LIN {X 0.007,Y -350.625,Z 530.640,A 0.000,B 0.000,C 90.000,E1 115.155} C_DIS
LIN {X -0.166,Y -363.454,Z 530.626,A 0.000,B 0.000,C 90.000,E1 112.770} C_DIS
LIN {X 0.046,Y -377.608,Z 530.613,A 0.000,B 0.000,C 90.000,E1 110.375} C_DIS
LIN {X 0.134,Y -393.193,Z 530.600,A 0.000,B 0.000,C 90.000,E1 108.055} C_DIS
LIN {X -0.144,Y -410.320,Z 530.588,A 0.000,B 0.000,C 90.000,E1 105.843} C_DIS
LIN {X -0.125,Y -429.118,Z 530.576,A 0.000,B 0.000,C 90.000,E1 103.647} C_DIS
LIN {X 0.160,Y -449.156,Z 530.564,A 0.000,B 0.000,C 90.000,E1 101.535} C_DIS
LIN {X -0.139,Y -469.752,Z 530.554,A 0.000,B 0.000,C 90.000,E1 99.670} C_DIS
LIN {X 0.073,Y -477.496,Z 530.550,A 0.000,B 0.000,C 90.000,E1 98.973} C_DIS
LIN {X 0.123,Y -479.452,Z 530.549,A 0.000,B 0.000,C 90.000,E1 98.746} C_DIS
LIN {X -0.005,Y -481.138,Z 530.547,A 0.000,B 0.000,C 90.000,E1 98.511} C_DIS
LIN {X -0.136,Y -482.404,Z 530.546,A 0.000,B 0.000,C 90.000,E1 98.276} C_DIS
LIN {X 0.031,Y -483.966,Z 530.543,A 0.000,B 0.000,C 90.000,E1 97.757} C_DIS
LIN {X 0.207,Y -484.472,Z 530.540,A 0.000,B 0.000,C 90.000,E1 97.239} C_DIS
LIN {X -0.087,Y -484.003,Z 530.538,A 0.000,B 0.000,C 90.000,E1 96.777} C_DIS
LIN {X 0.102,Y -482.486,Z 530.535,A 0.000,B 0.000,C 90.000,E1 96.258} C_DIS
LIN {X -0.070,Y -481.251,Z 530.533,A 0.000,B 0.000,C 90.000,E1 96.030} C_DIS
LIN {X -0.191,Y -479.606,Z 530.532,A 0.000,B 0.000,C 90.000,E1 95.796} C_DIS
LIN {X 0.087,Y -461.916,Z 530.519,A 0.000,B 0.000,C 90.000,E1 93.498} C_DIS
LIN {X 0.151,Y -451.298,Z 530.511,A 0.000,B 0.000,C 90.000,E1 91.949} C_DIS
LIN {X -0.041,Y -438.774,Z 530.499,A 0.000,B 0.000,C 90.000,E1 89.885} C_DIS
LIN {X 0.054,Y -429.143,Z 530.490,A 0.000,B 0.000,C 90.000,E1 88.282} C_DIS
LIN {X -0.197,Y -416.360,Z 530.479,A 0.000,B 0.000,C 90.000,E1 86.159} C_DIS
LIN {X 0.150,Y -403.728,Z 530.466,A 0.000,B 0.000,C 90.000,E1 83.913} C_DIS
LIN {X 0.177,Y -392.888,Z 530.455,A 0.000,B 0.000,C 90.000,E1 81.951} C_DIS
LIN {X 0.024,Y -381.992,Z 530.444,A 0.000,B 0.000,C 90.000,E1 79.982} C_DIS
LIN {X 0.133,Y -366.500,Z 530.428,A 0.000,B 0.000,C 90.000,E1 77.061} C_DIS
LIN {X 0.143,Y -357.922,Z 530.418,A 0.000,B 0.000,C 90.000,E1 75.283} C_DIS
LIN {X -0.016,Y -346.420,Z 530.403,A 0.000,B 0.000,C 90.000,E1 72.598} C_DIS
LIN {X 0.049,Y -335.338,Z 530.386,A 0.000,B 0.000,C 90.000,E1 69.518} C_DIS
LIN {X -0.030,Y -325.168,Z 530.369,A 0.000,B 0.000,C 90.000,E1 66.410} C_DIS
LIN {X -0.152,Y -317.591,Z 530.355,A 0.000,B 0.000,C 90.000,E1 63.896} C_DIS
LIN {X -0.045,Y -309.997,Z 530.341,A 0.000,B 0.000,C 90.000,E1 61.307} C_DIS
LIN {X 0.168,Y -302.402,Z 530.326,A 0.000,B 0.000,C 90.000,E1 58.663} C_DIS
LIN {X 0.004,Y -293.272,Z 530.308,A 0.000,B 0.000,C 90.000,E1 55.388} C_DIS
LIN {X -0.063,Y -286.330,Z 530.293,A 0.000,B 0.000,C 90.000,E1 52.718} C_DIS
LIN {X -0.042,Y -281.026,Z 530.281,A 0.000,B 0.000,C 90.000,E1 50.678} C_DIS
LIN {X 0.012,Y -277.267,Z 530.274,A 0.000,B 0.000,C 90.000,E1 49.299} C_DIS
LIN {X 0.024,Y -273.186,Z 530.266,A 0.000,B 0.000,C 90.000,E1 47.919} C_DIS
LIN {X 0.128,Y -266.584,Z 530.255,A 0.000,B 0.000,C 90.000,E1 45.810} C_DIS
LIN {X 0.076,Y -259.610,Z 530.243,A 0.000,B 0.000,C 90.000,E1 43.704} C_DIS
LIN {X 0.135,Y -249.136,Z 530.225,A 0.000,B 0.000,C 90.000,E1 40.458} C_DIS
LIN {X -0.025,Y -239.322,Z 530.207,A 0.000,B 0.000,C 90.000,E1 37.202} C_DIS
LIN {X 0.076,Y -231.432,Z 530.190,A 0.000,B 0.000,C 90.000,E1 34.199} C_DIS
LIN {X -0.073,Y -224.272,Z 530.173,A 0.000,B 0.000,C 90.000,E1 31.209} C_DIS
LIN {X 0.064,Y -217.981,Z 530.156,A 0.000,B 0.000,C 90.000,E1 28.103} C_DIS
LIN {X -0.070,Y -212.533,Z 530.139,A 0.000,B 0.000,C 90.000,E1 25.027} C_DIS
LIN {X 0.062,Y -207.862,Z 530.121,A 0.000,B 0.000,C 90.000,E1 21.844} C_DIS
LIN {X 0.037,Y -203.164,Z 530.099,A 0.000,B 0.000,C 90.000,E1 17.873} C_DIS
LIN {X -0.011,Y -198.859,Z 530.073,A 0.000,B 0.000,C 90.000,E1 13.063} C_DIS
LIN {X 0.096,Y -195.722,Z 530.041,A 0.000,B 0.000,C 90.000,E1 7.352} C_DIS
LIN {X 0.022,Y -196.744,Z 529.961,A 0.000,B 0.000,C 90.000,E1 352.996} C_DIS
LIN {X 0.044,Y -199.908,Z 529.934,A 0.000,B 0.000,C 90.000,E1 348.117} C_DIS
LIN {X -0.099,Y -204.347,Z 529.907,A 0.000,B 0.000,C 90.000,E1 343.323} C_DIS
LIN {X -0.047,Y -208.988,Z 529.885,A 0.000,B 0.000,C 90.000,E1 339.316} C_DIS
LIN {X -0.013,Y -214.345,Z 529.863,A 0.000,B 0.000,C 90.000,E1 335.357} C_DIS
LIN {X 0.053,Y -220.253,Z 529.841,A 0.000,B 0.000,C 90.000,E1 331.435} C_DIS
LIN {X 0.050,Y -226.713,Z 529.820,A 0.000,B 0.000,C 90.000,E1 327.582} C_DIS
LIN {X 0.037,Y -233.852,Z 529.799,A 0.000,B 0.000,C 90.000,E1 323.783} C_DIS
LIN {X -0.099,Y -241.522,Z 529.778,A 0.000,B 0.000,C 90.000,E1 320.070} C_DIS
LIN {X -0.078,Y -250.132,Z 529.758,A 0.000,B 0.000,C 90.000,E1 316.377} C_DIS
LIN {X -0.146,Y -259.993,Z 529.737,A 0.000,B 0.000,C 90.000,E1 312.771} C_DIS
LIN {X -0.008,Y -271.110,Z 529.718,A 0.000,B 0.000,C 90.000,E1 309.197} C_DIS
LIN {X 0.019,Y -283.470,Z 529.698,A 0.000,B 0.000,C 90.000,E1 305.724} C_DIS
LIN {X 0.018,Y -297.205,Z 529.680,A 0.000,B 0.000,C 90.000,E1 302.339} C_DIS
LIN {X 0.091,Y -312.087,Z 529.661,A 0.000,B 0.000,C 90.000,E1 299.027} C_DIS
LIN {X -0.031,Y -326.602,Z 529.645,A 0.000,B 0.000,C 90.000,E1 296.155} C_DIS
LIN {X -0.104,Y -335.578,Z 529.637,A 0.000,B 0.000,C 90.000,E1 294.591} C_DIS
LIN {X -0.001,Y -349.328,Z 529.625,A 0.000,B 0.000,C 90.000,E1 292.408} C_DIS
LIN {X -0.061,Y -364.291,Z 529.613,A 0.000,B 0.000,C 90.000,E1 290.301} C_DIS
LIN {X 0.072,Y -385.334,Z 529.598,A 0.000,B 0.000,C 90.000,E1 287.638} C_DIS
LIN {X -0.069,Y -402.321,Z 529.587,A 0.000,B 0.000,C 90.000,E1 285.662} C_DIS
LIN {X -0.186,Y -417.218,Z 529.578,A 0.000,B 0.000,C 90.000,E1 284.008} C_DIS
LIN {X -0.176,Y -429.390,Z 529.570,A 0.000,B 0.000,C 90.000,E1 282.647} C_DIS
LIN {X -0.114,Y -441.000,Z 529.563,A 0.000,B 0.000,C 90.000,E1 281.299} C_DIS
LIN {X 0.019,Y -447.666,Z 529.558,A 0.000,B 0.000,C 90.000,E1 280.489} C_DIS
LIN {X 0.026,Y -455.859,Z 529.552,A 0.000,B 0.000,C 90.000,E1 279.443} C_DIS
LIN {X 0.132,Y -463.364,Z 529.547,A 0.000,B 0.000,C 90.000,E1 278.398} C_DIS
LIN {X 0.017,Y -468.372,Z 529.542,A 0.000,B 0.000,C 90.000,E1 277.644} C_DIS
LIN {X -0.052,Y -472.900,Z 529.538,A 0.000,B 0.000,C 90.000,E1 276.891} C_DIS
LIN {X -0.144,Y -476.941,Z 529.534,A 0.000,B 0.000,C 90.000,E1 276.144} C_DIS
LIN {X -0.146,Y -480.361,Z 529.530,A 0.000,B 0.000,C 90.000,E1 275.391} C_DIS
LIN {X -0.171,Y -483.141,Z 529.526,A 0.000,B 0.000,C 90.000,E1 274.645} C_DIS
LIN {X -0.039,Y -484.544,Z 529.523,A 0.000,B 0.000,C 90.000,E1 274.131} C_DIS
LIN {X 0.140,Y -485.652,Z 529.520,A 0.000,B 0.000,C 90.000,E1 273.612} C_DIS
LIN {X -0.161,Y -486.454,Z 529.517,A 0.000,B 0.000,C 90.000,E1 273.151} C_DIS
LIN {X 0.002,Y -486.937,Z 529.515,A 0.000,B 0.000,C 90.000,E1 272.636} C_DIS
LIN {X 0.173,Y -487.084,Z 529.512,A 0.000,B 0.000,C 90.000,E1 272.121} C_DIS
LIN {X -0.122,Y -486.839,Z 529.509,A 0.000,B 0.000,C 90.000,E1 271.661} C_DIS
LIN {X 0.053,Y -486.202,Z 529.506,A 0.000,B 0.000,C 90.000,E1 271.146} C_DIS
LIN {X 0.229,Y -485.150,Z 529.504,A 0.000,B 0.000,C 90.000,E1 270.630} C_DIS
LIN {X -0.084,Y -483.586,Z 529.501,A 0.000,B 0.000,C 90.000,E1 270.172} C_DIS
LIN {X 0.082,Y -481.379,Z 529.498,A 0.000,B 0.000,C 90.000,E1 269.656} C_DIS
LIN {X 0.231,Y -478.423,Z 529.495,A 0.000,B 0.000,C 90.000,E1 269.141} C_DIS
LIN {X -0.113,Y -474.579,Z 529.493,A 0.000,B 0.000,C 90.000,E1 268.682} C_DIS
LIN {X 0.015,Y -469.635,Z 529.490,A 0.000,B 0.000,C 90.000,E1 268.165} C_DIS
LIN {X -0.092,Y -466.805,Z 529.488,A 0.000,B 0.000,C 90.000,E1 267.936} C_DIS
LIN {X -0.197,Y -463.629,Z 529.487,A 0.000,B 0.000,C 90.000,E1 267.707} C_DIS
LIN {X -0.022,Y -460.564,Z 529.486,A 0.000,B 0.000,C 90.000,E1 267.478} C_DIS
LIN {X 0.152,Y -453.814,Z 529.484,A 0.000,B 0.000,C 90.000,E1 267.078} C_DIS
LIN {X -0.011,Y -446.799,Z 529.482,A 0.000,B 0.000,C 90.000,E1 266.788} C_DIS
LIN {X -0.202,Y -439.772,Z 529.481,A 0.000,B 0.000,C 90.000,E1 266.560} C_DIS
LIN {X -0.051,Y -432.358,Z 529.480,A 0.000,B 0.000,C 90.000,E1 266.331} C_DIS
LIN {X 0.005,Y -424.212,Z 529.479,A 0.000,B 0.000,C 90.000,E1 266.159} C_DIS
LIN {X -0.004,Y -414.402,Z 529.478,A 0.000,B 0.000,C 90.000,E1 266.045} C_DIS
LIN {X 0.134,Y -407.149,Z 529.478,A 0.000,B 0.000,C 90.000,E1 265.988} C_DIS
LIN {X 0.040,Y -180.920,Z 529.478,A 0.000,B 0.000,C 90.000,E1 265.988} C_DIS
LIN {X -0.084,Y -180.857,Z 529.472,A 0.000,B 0.000,C 90.000,E1 265.008} C_DIS
LIN {X -0.005,Y -178.910,Z 529.443,A 0.000,B 0.000,C 90.000,E1 259.746} C_DIS
LIN {X 0.076,Y -175.954,Z 529.415,A 0.000,B 0.000,C 90.000,E1 254.629} C_DIS
LIN {X 0.022,Y -175.423,Z 529.410,A 0.000,B 0.000,C 90.000,E1 253.795} C_DIS
LIN {X 0.025,Y -172.184,Z 529.386,A 0.000,B 0.000,C 90.000,E1 249.518} C_DIS
LIN {X 0.063,Y -171.656,Z 529.381,A 0.000,B 0.000,C 90.000,E1 248.646} C_DIS
LIN {X 0.057,Y -167.880,Z 529.357,A 0.000,B 0.000,C 90.000,E1 244.332} C_DIS
LIN {X 0.001,Y -166.615,Z 529.348,A 0.000,B 0.000,C 90.000,E1 242.615} C_DIS
LIN {X -0.006,Y -162.602,Z 529.324,A 0.000,B 0.000,C 90.000,E1 238.250} C_DIS
LIN {X -0.032,Y -161.288,Z 529.314,A 0.000,B 0.000,C 90.000,E1 236.501} C_DIS
LIN {X 0.003,Y -157.287,Z 529.289,A 0.000,B 0.000,C 90.000,E1 232.065} C_DIS
LIN {X 0.026,Y -156.004,Z 529.279,A 0.000,B 0.000,C 90.000,E1 230.275} C_DIS
LIN {X -0.014,Y -152.262,Z 529.254,A 0.000,B 0.000,C 90.000,E1 225.810} C_DIS
LIN {X 0.008,Y -150.500,Z 529.239,A 0.000,B 0.000,C 90.000,E1 223.095} C_DIS
LIN {X 0.038,Y -147.224,Z 529.214,A 0.000,B 0.000,C 90.000,E1 218.543} C_DIS
LIN {X 0.008,Y -145.247,Z 529.194,A 0.000,B 0.000,C 90.000,E1 214.898} C_DIS
LIN {X -0.076,Y -142.364,Z 529.163,A 0.000,B 0.000,C 90.000,E1 209.411} C_DIS
LIN {X 0.045,Y -141.750,Z 529.153,A 0.000,B 0.000,C 90.000,E1 207.513} C_DIS
LIN {X -0.029,Y -139.494,Z 529.117,A 0.000,B 0.000,C 90.000,E1 201.046} C_DIS
LIN {X 0.007,Y -138.997,Z 529.101,A 0.000,B 0.000,C 90.000,E1 198.236} C_DIS
LIN {X -0.036,Y -138.338,Z 529.055,A 0.000,B 0.000,C 90.000,E1 189.849} C_DIS
LIN {X -0.014,Y -139.412,Z 529.008,A 0.000,B 0.000,C 90.000,E1 181.432} C_DIS
LIN {X 0.040,Y -141.325,Z 528.972,A 0.000,B 0.000,C 90.000,E1 174.894} C_DIS
LIN {X -0.003,Y -142.683,Z 528.956,A 0.000,B 0.000,C 90.000,E1 172.129} C_DIS
LIN {X -0.024,Y -145.042,Z 528.931,A 0.000,B 0.000,C 90.000,E1 167.521} C_DIS
LIN {X -0.026,Y -147.667,Z 528.910,A 0.000,B 0.000,C 90.000,E1 163.850} C_DIS
LIN {X 0.009,Y -150.309,Z 528.890,A 0.000,B 0.000,C 90.000,E1 160.188} C_DIS
LIN {X 0.020,Y -153.720,Z 528.870,A 0.000,B 0.000,C 90.000,E1 156.561} C_DIS
LIN {X -0.067,Y -157.134,Z 528.850,A 0.000,B 0.000,C 90.000,E1 152.999} C_DIS
LIN {X 0.009,Y -161.281,Z 528.830,A 0.000,B 0.000,C 90.000,E1 149.410} C_DIS
LIN {X 0.026,Y -164.397,Z 528.815,A 0.000,B 0.000,C 90.000,E1 146.755} C_DIS
LIN {X 0.023,Y -169.076,Z 528.796,A 0.000,B 0.000,C 90.000,E1 143.256} C_DIS
LIN {X -0.026,Y -171.634,Z 528.786,A 0.000,B 0.000,C 90.000,E1 141.537} C_DIS
LIN {X 0.021,Y -176.595,Z 528.767,A 0.000,B 0.000,C 90.000,E1 138.081} C_DIS
LIN {X -0.107,Y -180.893,Z 528.753,A 0.000,B 0.000,C 90.000,E1 135.567} C_DIS
LIN {X 0.015,Y -186.308,Z 528.734,A 0.000,B 0.000,C 90.000,E1 132.162} C_DIS
LIN {X 0.076,Y -191.412,Z 528.719,A 0.000,B 0.000,C 90.000,E1 129.358} C_DIS
LIN {X -0.043,Y -192.207,Z 528.716,A 0.000,B 0.000,C 90.000,E1 128.910} C_DIS
LIN {X -0.099,Y -289.108,Z 528.716,A 0.000,B 0.000,C 90.000,E1 128.910} C_DIS
LIN {X 0.061,Y -291.712,Z 528.716,A 0.000,B 0.000,C 90.000,E1 128.830} C_DIS
LIN {X 0.026,Y -294.579,Z 528.715,A 0.000,B 0.000,C 90.000,E1 128.705} C_DIS
LIN {X 0.024,Y -298.101,Z 528.713,A 0.000,B 0.000,C 90.000,E1 128.418} C_DIS
LIN {X 0.036,Y -301.731,Z 528.711,A 0.000,B 0.000,C 90.000,E1 127.935} C_DIS
LIN {X 0.036,Y -303.492,Z 528.709,A 0.000,B 0.000,C 90.000,E1 127.604} C_DIS
LIN {X -0.022,Y -304.870,Z 528.707,A 0.000,B 0.000,C 90.000,E1 127.282} C_DIS
LIN {X -0.001,Y -310.679,Z 528.696,A 0.000,B 0.000,C 90.000,E1 125.311} C_DIS
LIN {X -0.024,Y -321.264,Z 528.678,A 0.000,B 0.000,C 90.000,E1 122.084} C_DIS
LIN {X 0.130,Y -332.150,Z 528.662,A 0.000,B 0.000,C 90.000,E1 119.205} C_DIS
LIN {X -0.051,Y -344.433,Z 528.647,A 0.000,B 0.000,C 90.000,E1 116.437} C_DIS
LIN {X -0.082,Y -356.610,Z 528.633,A 0.000,B 0.000,C 90.000,E1 114.003} C_DIS
LIN {X 0.082,Y -370.065,Z 528.620,A 0.000,B 0.000,C 90.000,E1 111.589} C_DIS
LIN {X -0.022,Y -384.893,Z 528.607,A 0.000,B 0.000,C 90.000,E1 109.268} C_DIS
LIN {X -0.005,Y -401.205,Z 528.594,A 0.000,B 0.000,C 90.000,E1 106.985} C_DIS
LIN {X -0.087,Y -419.119,Z 528.582,A 0.000,B 0.000,C 90.000,E1 104.773} C_DIS
LIN {X 0.140,Y -438.656,Z 528.570,A 0.000,B 0.000,C 90.000,E1 102.591} C_DIS
LIN {X 0.136,Y -458.972,Z 528.559,A 0.000,B 0.000,C 90.000,E1 100.602} C_DIS
LIN {X -0.122,Y -477.137,Z 528.550,A 0.000,B 0.000,C 90.000,E1 99.029} C_DIS
LIN {X -0.077,Y -479.223,Z 528.549,A 0.000,B 0.000,C 90.000,E1 98.803} C_DIS
LIN {X -0.207,Y -481.005,Z 528.547,A 0.000,B 0.000,C 90.000,E1 98.568} C_DIS
LIN {X 0.138,Y -482.344,Z 528.546,A 0.000,B 0.000,C 90.000,E1 98.276} C_DIS
LIN {X -0.175,Y -484.021,Z 528.543,A 0.000,B 0.000,C 90.000,E1 97.814} C_DIS
LIN {X 0.001,Y -484.625,Z 528.541,A 0.000,B 0.000,C 90.000,E1 97.296} C_DIS
LIN {X 0.187,Y -484.254,Z 528.538,A 0.000,B 0.000,C 90.000,E1 96.777} C_DIS
LIN {X -0.104,Y -482.849,Z 528.535,A 0.000,B 0.000,C 90.000,E1 96.315} C_DIS
LIN {X 0.203,Y -481.685,Z 528.534,A 0.000,B 0.000,C 90.000,E1 96.030} C_DIS
LIN {X 0.083,Y -480.128,Z 528.532,A 0.000,B 0.000,C 90.000,E1 95.796} C_DIS
LIN {X 0.157,Y -460.553,Z 528.518,A 0.000,B 0.000,C 90.000,E1 93.269} C_DIS
LIN {X 0.212,Y -450.047,Z 528.510,A 0.000,B 0.000,C 90.000,E1 91.718} C_DIS
LIN {X -0.201,Y -439.126,Z 528.500,A 0.000,B 0.000,C 90.000,E1 89.943} C_DIS
LIN {X 0.063,Y -427.874,Z 528.489,A 0.000,B 0.000,C 90.000,E1 88.051} C_DIS
LIN {X 0.210,Y -415.100,Z 528.477,A 0.000,B 0.000,C 90.000,E1 85.869} C_DIS
LIN {X 0.079,Y -402.485,Z 528.465,A 0.000,B 0.000,C 90.000,E1 83.685} C_DIS
LIN {X 0.071,Y -391.630,Z 528.454,A 0.000,B 0.000,C 90.000,E1 81.724} C_DIS
LIN {X -0.040,Y -380.732,Z 528.443,A 0.000,B 0.000,C 90.000,E1 79.746} C_DIS
LIN {X 0.078,Y -362.338,Z 528.424,A 0.000,B 0.000,C 90.000,E1 76.228} C_DIS
LIN {X -0.096,Y -351.588,Z 528.410,A 0.000,B 0.000,C 90.000,E1 73.866} C_DIS
LIN {X 0.089,Y -343.134,Z 528.398,A 0.000,B 0.000,C 90.000,E1 71.710} C_DIS
LIN {X -0.041,Y -331.364,Z 528.380,A 0.000,B 0.000,C 90.000,E1 68.337} C_DIS
LIN {X 0.060,Y -321.469,Z 528.362,A 0.000,B 0.000,C 90.000,E1 65.177} C_DIS
LIN {X 0.116,Y -315.842,Z 528.352,A 0.000,B 0.000,C 90.000,E1 63.256} C_DIS
LIN {X -0.099,Y -308.215,Z 528.337,A 0.000,B 0.000,C 90.000,E1 60.717} C_DIS
LIN {X 0.065,Y -300.615,Z 528.323,A 0.000,B 0.000,C 90.000,E1 58.074} C_DIS
LIN {X 0.007,Y -291.582,Z 528.304,A 0.000,B 0.000,C 90.000,E1 54.769} C_DIS
LIN {X 0.066,Y -284.646,Z 528.289,A 0.000,B 0.000,C 90.000,E1 52.065} C_DIS
LIN {X 0.015,Y -279.246,Z 528.278,A 0.000,B 0.000,C 90.000,E1 50.033} C_DIS
LIN {X -0.127,Y -275.337,Z 528.270,A 0.000,B 0.000,C 90.000,E1 48.690} C_DIS
LIN {X -0.137,Y -271.113,Z 528.263,A 0.000,B 0.000,C 90.000,E1 47.310} C_DIS
LIN {X -0.143,Y -265.514,Z 528.253,A 0.000,B 0.000,C 90.000,E1 45.567} C_DIS
LIN {X -0.021,Y -258.491,Z 528.241,A 0.000,B 0.000,C 90.000,E1 43.419} C_DIS
LIN {X 0.022,Y -248.070,Z 528.223,A 0.000,B 0.000,C 90.000,E1 40.172} C_DIS
LIN {X 0.036,Y -239.368,Z 528.207,A 0.000,B 0.000,C 90.000,E1 37.237} C_DIS
LIN {X -0.045,Y -231.492,Z 528.190,A 0.000,B 0.000,C 90.000,E1 34.278} C_DIS
LIN {X -0.069,Y -224.332,Z 528.174,A 0.000,B 0.000,C 90.000,E1 31.258} C_DIS
LIN {X 0.064,Y -218.015,Z 528.156,A 0.000,B 0.000,C 90.000,E1 28.153} C_DIS
LIN {X -0.076,Y -212.566,Z 528.139,A 0.000,B 0.000,C 90.000,E1 25.079} C_DIS
LIN {X 0.053,Y -207.885,Z 528.122,A 0.000,B 0.000,C 90.000,E1 21.897} C_DIS
LIN {X -0.038,Y -203.189,Z 528.100,A 0.000,B 0.000,C 90.000,E1 17.946} C_DIS
LIN {X -0.027,Y -198.863,Z 528.073,A 0.000,B 0.000,C 90.000,E1 13.119} C_DIS
LIN {X 0.077,Y -195.705,Z 528.041,A 0.000,B 0.000,C 90.000,E1 7.409} C_DIS
LIN {X 0.019,Y -196.653,Z 527.961,A 0.000,B 0.000,C 90.000,E1 352.996} C_DIS
LIN {X 0.037,Y -199.811,Z 527.934,A 0.000,B 0.000,C 90.000,E1 348.117} C_DIS
LIN {X -0.110,Y -204.250,Z 527.907,A 0.000,B 0.000,C 90.000,E1 343.323} C_DIS
LIN {X -0.061,Y -208.893,Z 527.885,A 0.000,B 0.000,C 90.000,E1 339.316} C_DIS
LIN {X -0.031,Y -214.236,Z 527.863,A 0.000,B 0.000,C 90.000,E1 335.357} C_DIS
LIN {X 0.031,Y -220.166,Z 527.841,A 0.000,B 0.000,C 90.000,E1 331.435} C_DIS
LIN {X 0.026,Y -226.620,Z 527.820,A 0.000,B 0.000,C 90.000,E1 327.582} C_DIS
LIN {X 0.010,Y -233.769,Z 527.799,A 0.000,B 0.000,C 90.000,E1 323.783} C_DIS
LIN {X 0.024,Y -241.448,Z 527.778,A 0.000,B 0.000,C 90.000,E1 320.033} C_DIS
LIN {X -0.113,Y -250.080,Z 527.758,A 0.000,B 0.000,C 90.000,E1 316.377} C_DIS
LIN {X -0.023,Y -258.919,Z 527.739,A 0.000,B 0.000,C 90.000,E1 313.095} C_DIS
LIN {X -0.121,Y -269.921,Z 527.720,A 0.000,B 0.000,C 90.000,E1 309.564} C_DIS
LIN {X -0.136,Y -282.164,Z 527.700,A 0.000,B 0.000,C 90.000,E1 306.091} C_DIS
LIN {X -0.019,Y -295.786,Z 527.682,A 0.000,B 0.000,C 90.000,E1 302.673} C_DIS
LIN {X 0.155,Y -310.524,Z 527.663,A 0.000,B 0.000,C 90.000,E1 299.333} C_DIS
LIN {X -0.080,Y -326.591,Z 527.645,A 0.000,B 0.000,C 90.000,E1 296.155} C_DIS
LIN {X -0.154,Y -335.584,Z 527.636,A 0.000,B 0.000,C 90.000,E1 294.591} C_DIS
LIN {X 0.095,Y -351.378,Z 527.623,A 0.000,B 0.000,C 90.000,E1 292.078} C_DIS
LIN {X -0.046,Y -366.538,Z 527.611,A 0.000,B 0.000,C 90.000,E1 289.993} C_DIS
LIN {X 0.026,Y -387.760,Z 527.596,A 0.000,B 0.000,C 90.000,E1 287.347} C_DIS
LIN {X -0.051,Y -404.810,Z 527.585,A 0.000,B 0.000,C 90.000,E1 285.371} C_DIS
LIN {X -0.018,Y -419.735,Z 527.576,A 0.000,B 0.000,C 90.000,E1 283.703} C_DIS
LIN {X 0.043,Y -431.720,Z 527.569,A 0.000,B 0.000,C 90.000,E1 282.355} C_DIS
LIN {X 0.154,Y -443.239,Z 527.561,A 0.000,B 0.000,C 90.000,E1 281.007} C_DIS
LIN {X -0.137,Y -449.792,Z 527.557,A 0.000,B 0.000,C 90.000,E1 280.254} C_DIS
LIN {X -0.108,Y -457.858,Z 527.551,A 0.000,B 0.000,C 90.000,E1 279.208} C_DIS
LIN {X 0.191,Y -463.412,Z 527.547,A 0.000,B 0.000,C 90.000,E1 278.398} C_DIS
LIN {X 0.078,Y -468.442,Z 527.543,A 0.000,B 0.000,C 90.000,E1 277.644} C_DIS
LIN {X -0.203,Y -474.387,Z 527.537,A 0.000,B 0.000,C 90.000,E1 276.663} C_DIS
LIN {X 0.249,Y -478.248,Z 527.533,A 0.000,B 0.000,C 90.000,E1 275.853} C_DIS
LIN {X 0.210,Y -481.467,Z 527.529,A 0.000,B 0.000,C 90.000,E1 275.106} C_DIS
LIN {X -0.107,Y -483.226,Z 527.526,A 0.000,B 0.000,C 90.000,E1 274.645} C_DIS
LIN {X 0.026,Y -484.669,Z 527.523,A 0.000,B 0.000,C 90.000,E1 274.131} C_DIS
LIN {X 0.206,Y -485.766,Z 527.520,A 0.000,B 0.000,C 90.000,E1 273.612} C_DIS
LIN {X -0.122,Y -486.559,Z 527.517,A 0.000,B 0.000,C 90.000,E1 273.154} C_DIS
LIN {X 0.069,Y -487.048,Z 527.515,A 0.000,B 0.000,C 90.000,E1 272.636} C_DIS
LIN {X -0.245,Y -487.209,Z 527.512,A 0.000,B 0.000,C 90.000,E1 272.178} C_DIS
LIN {X -0.054,Y -486.949,Z 527.509,A 0.000,B 0.000,C 90.000,E1 271.661} C_DIS
LIN {X 0.123,Y -486.313,Z 527.506,A 0.000,B 0.000,C 90.000,E1 271.146} C_DIS
LIN {X -0.188,Y -485.245,Z 527.504,A 0.000,B 0.000,C 90.000,E1 270.688} C_DIS
LIN {X -0.014,Y -483.677,Z 527.501,A 0.000,B 0.000,C 90.000,E1 270.172} C_DIS
LIN {X 0.152,Y -481.499,Z 527.498,A 0.000,B 0.000,C 90.000,E1 269.656} C_DIS
LIN {X -0.177,Y -478.524,Z 527.495,A 0.000,B 0.000,C 90.000,E1 269.198} C_DIS
LIN {X 0.129,Y -476.771,Z 527.494,A 0.000,B 0.000,C 90.000,E1 268.912} C_DIS
LIN {X -0.221,Y -472.351,Z 527.491,A 0.000,B 0.000,C 90.000,E1 268.453} C_DIS
LIN {X 0.085,Y -469.779,Z 527.490,A 0.000,B 0.000,C 90.000,E1 268.165} C_DIS
LIN {X -0.032,Y -466.971,Z 527.489,A 0.000,B 0.000,C 90.000,E1 267.936} C_DIS
LIN {X -0.147,Y -463.777,Z 527.487,A 0.000,B 0.000,C 90.000,E1 267.707} C_DIS
LIN {X 0.200,Y -457.215,Z 527.485,A 0.000,B 0.000,C 90.000,E1 267.249} C_DIS
LIN {X 0.153,Y -450.105,Z 527.483,A 0.000,B 0.000,C 90.000,E1 266.906} C_DIS
LIN {X -0.191,Y -443.079,Z 527.481,A 0.000,B 0.000,C 90.000,E1 266.674} C_DIS
LIN {X -0.192,Y -435.942,Z 527.480,A 0.000,B 0.000,C 90.000,E1 266.445} C_DIS
LIN {X 0.123,Y -428.327,Z 527.479,A 0.000,B 0.000,C 90.000,E1 266.216} C_DIS
LIN {X -0.083,Y -419.441,Z 527.478,A 0.000,B 0.000,C 90.000,E1 266.102} C_DIS
LIN {X 0.142,Y -408.334,Z 527.478,A 0.000,B 0.000,C 90.000,E1 265.988} C_DIS
LIN {X 0.095,Y -405.887,Z 527.478,A 0.000,B 0.000,C 90.000,E1 265.988} C_DIS
LIN {X 0.023,Y -180.920,Z 527.478,A 0.000,B 0.000,C 90.000,E1 265.988} C_DIS
LIN {X 0.080,Y -180.856,Z 527.472,A 0.000,B 0.000,C 90.000,E1 264.951} C_DIS
LIN {X -0.021,Y -178.908,Z 527.443,A 0.000,B 0.000,C 90.000,E1 259.746} C_DIS
LIN {X 0.060,Y -175.952,Z 527.415,A 0.000,B 0.000,C 90.000,E1 254.629} C_DIS
LIN {X 0.006,Y -175.418,Z 527.410,A 0.000,B 0.000,C 90.000,E1 253.795} C_DIS
LIN {X 0.008,Y -172.180,Z 527.386,A 0.000,B 0.000,C 90.000,E1 249.518} C_DIS
LIN {X 0.048,Y -171.651,Z 527.381,A 0.000,B 0.000,C 90.000,E1 248.646} C_DIS
LIN {X 0.042,Y -167.876,Z 527.357,A 0.000,B 0.000,C 90.000,E1 244.332} C_DIS
LIN {X -0.015,Y -166.611,Z 527.348,A 0.000,B 0.000,C 90.000,E1 242.615} C_DIS
LIN {X -0.021,Y -162.599,Z 527.324,A 0.000,B 0.000,C 90.000,E1 238.250} C_DIS
LIN {X -0.047,Y -161.283,Z 527.314,A 0.000,B 0.000,C 90.000,E1 236.501} C_DIS
LIN {X -0.012,Y -157.282,Z 527.289,A 0.000,B 0.000,C 90.000,E1 232.065} C_DIS
LIN {X 0.011,Y -156.000,Z 527.279,A 0.000,B 0.000,C 90.000,E1 230.275} C_DIS
LIN {X -0.029,Y -152.258,Z 527.254,A 0.000,B 0.000,C 90.000,E1 225.810} C_DIS
LIN {X -0.006,Y -150.496,Z 527.239,A 0.000,B 0.000,C 90.000,E1 223.095} C_DIS
LIN {X 0.024,Y -147.221,Z 527.214,A 0.000,B 0.000,C 90.000,E1 218.543} C_DIS
LIN {X -0.007,Y -145.243,Z 527.194,A 0.000,B 0.000,C 90.000,E1 214.898} C_DIS
LIN {X -0.090,Y -142.362,Z 527.163,A 0.000,B 0.000,C 90.000,E1 209.411} C_DIS
LIN {X 0.031,Y -141.748,Z 527.153,A 0.000,B 0.000,C 90.000,E1 207.513} C_DIS
LIN {X -0.043,Y -139.492,Z 527.117,A 0.000,B 0.000,C 90.000,E1 201.046} C_DIS
LIN {X -0.006,Y -138.996,Z 527.101,A 0.000,B 0.000,C 90.000,E1 198.236} C_DIS
LIN {X -0.050,Y -138.337,Z 527.055,A 0.000,B 0.000,C 90.000,E1 189.849} C_DIS
LIN {X -0.028,Y -139.414,Z 527.008,A 0.000,B 0.000,C 90.000,E1 181.432} C_DIS
LIN {X 0.026,Y -141.328,Z 526.972,A 0.000,B 0.000,C 90.000,E1 174.894} C_DIS
LIN {X -0.017,Y -142.685,Z 526.956,A 0.000,B 0.000,C 90.000,E1 172.129} C_DIS
LIN {X -0.037,Y -145.045,Z 526.931,A 0.000,B 0.000,C 90.000,E1 167.521} C_DIS
LIN {X -0.040,Y -147.671,Z 526.910,A 0.000,B 0.000,C 90.000,E1 163.850} C_DIS
LIN {X -0.006,Y -150.313,Z 526.890,A 0.000,B 0.000,C 90.000,E1 160.188} C_DIS
LIN {X 0.067,Y -153.726,Z 526.870,A 0.000,B 0.000,C 90.000,E1 156.538} C_DIS
LIN {X -0.082,Y -157.139,Z 526.850,A 0.000,B 0.000,C 90.000,E1 152.999} C_DIS
LIN {X -0.006,Y -161.287,Z 526.830,A 0.000,B 0.000,C 90.000,E1 149.410} C_DIS
LIN {X 0.011,Y -164.403,Z 526.815,A 0.000,B 0.000,C 90.000,E1 146.755} C_DIS
LIN {X 0.008,Y -169.084,Z 526.796,A 0.000,B 0.000,C 90.000,E1 143.256} C_DIS
LIN {X -0.042,Y -171.641,Z 526.786,A 0.000,B 0.000,C 90.000,E1 141.537} C_DIS
LIN {X 0.005,Y -176.603,Z 526.767,A 0.000,B 0.000,C 90.000,E1 138.081} C_DIS
LIN {X 0.007,Y -180.901,Z 526.753,A 0.000,B 0.000,C 90.000,E1 135.526} C_DIS
LIN {X -0.002,Y -186.317,Z 526.734,A 0.000,B 0.000,C 90.000,E1 132.162} C_DIS
LIN {X 0.058,Y -191.420,Z 526.719,A 0.000,B 0.000,C 90.000,E1 129.358} C_DIS
LIN {X -0.085,Y -192.228,Z 526.716,A 0.000,B 0.000,C 90.000,E1 128.910} C_DIS
LIN {X -0.158,Y -289.363,Z 526.716,A 0.000,B 0.000,C 90.000,E1 128.910} C_DIS
LIN {X 0.035,Y -291.563,Z 526.716,A 0.000,B 0.000,C 90.000,E1 128.830} C_DIS
LIN {X 0.014,Y -295.030,Z 526.715,A 0.000,B 0.000,C 90.000,E1 128.669} C_DIS
LIN {X -0.036,Y -298.461,Z 526.713,A 0.000,B 0.000,C 90.000,E1 128.382} C_DIS
LIN {X -0.099,Y -302.097,Z 526.710,A 0.000,B 0.000,C 90.000,E1 127.890} C_DIS
LIN {X 0.086,Y -303.777,Z 526.709,A 0.000,B 0.000,C 90.000,E1 127.523} C_DIS
LIN {X -0.155,Y -305.095,Z 526.707,A 0.000,B 0.000,C 90.000,E1 127.237} C_DIS
LIN {X -0.040,Y -315.984,Z 526.687,A 0.000,B 0.000,C 90.000,E1 123.627} C_DIS
LIN {X 0.116,Y -326.170,Z 526.671,A 0.000,B 0.000,C 90.000,E1 120.718} C_DIS
LIN {X 0.079,Y -337.695,Z 526.655,A 0.000,B 0.000,C 90.000,E1 117.897} C_DIS
LIN {X -0.103,Y -350.668,Z 526.640,A 0.000,B 0.000,C 90.000,E1 115.155} C_DIS
LIN {X 0.058,Y -363.505,Z 526.626,A 0.000,B 0.000,C 90.000,E1 112.717} C_DIS
LIN {X -0.068,Y -377.670,Z 526.613,A 0.000,B 0.000,C 90.000,E1 110.375} C_DIS
LIN {X 0.016,Y -393.266,Z 526.600,A 0.000,B 0.000,C 90.000,E1 108.055} C_DIS
LIN {X 0.128,Y -410.404,Z 526.588,A 0.000,B 0.000,C 90.000,E1 105.788} C_DIS
LIN {X 0.167,Y -429.214,Z 526.576,A 0.000,B 0.000,C 90.000,E1 103.592} C_DIS
LIN {X 0.038,Y -449.257,Z 526.564,A 0.000,B 0.000,C 90.000,E1 101.535} C_DIS
LIN {X 0.205,Y -469.857,Z 526.554,A 0.000,B 0.000,C 90.000,E1 99.613} C_DIS
LIN {X -0.044,Y -477.630,Z 526.550,A 0.000,B 0.000,C 90.000,E1 98.973} C_DIS
LIN {X 0.006,Y -479.632,Z 526.549,A 0.000,B 0.000,C 90.000,E1 98.746} C_DIS
LIN {X -0.122,Y -481.357,Z 526.547,A 0.000,B 0.000,C 90.000,E1 98.511} C_DIS
LIN {X 0.224,Y -482.653,Z 526.546,A 0.000,B 0.000,C 90.000,E1 98.219} C_DIS
LIN {X -0.085,Y -484.264,Z 526.543,A 0.000,B 0.000,C 90.000,E1 97.757} C_DIS
LIN {X 0.093,Y -484.813,Z 526.540,A 0.000,B 0.000,C 90.000,E1 97.239} C_DIS
LIN {X -0.201,Y -484.386,Z 526.538,A 0.000,B 0.000,C 90.000,E1 96.777} C_DIS
LIN {X -0.009,Y -482.914,Z 526.535,A 0.000,B 0.000,C 90.000,E1 96.258} C_DIS
LIN {X -0.130,Y -481.708,Z 526.533,A 0.000,B 0.000,C 90.000,E1 96.024} C_DIS
LIN {X 0.179,Y -480.098,Z 526.532,A 0.000,B 0.000,C 90.000,E1 95.739} C_DIS
LIN {X -0.211,Y -460.462,Z 526.518,A 0.000,B 0.000,C 90.000,E1 93.269} C_DIS
LIN {X -0.149,Y -449.933,Z 526.509,A 0.000,B 0.000,C 90.000,E1 91.718} C_DIS
LIN {X -0.117,Y -438.979,Z 526.499,A 0.000,B 0.000,C 90.000,E1 89.885} C_DIS
LIN {X 0.142,Y -427.710,Z 526.489,A 0.000,B 0.000,C 90.000,E1 87.993} C_DIS
LIN {X -0.042,Y -413.333,Z 526.475,A 0.000,B 0.000,C 90.000,E1 85.584} C_DIS
LIN {X -0.168,Y -400.748,Z 526.463,A 0.000,B 0.000,C 90.000,E1 83.394} C_DIS
LIN {X 0.185,Y -391.440,Z 526.454,A 0.000,B 0.000,C 90.000,E1 81.659} C_DIS
LIN {X 0.009,Y -380.542,Z 526.443,A 0.000,B 0.000,C 90.000,E1 79.690} C_DIS
LIN {X 0.113,Y -362.153,Z 526.423,A 0.000,B 0.000,C 90.000,E1 76.172} C_DIS
LIN {X 0.029,Y -351.410,Z 526.410,A 0.000,B 0.000,C 90.000,E1 73.795} C_DIS
LIN {X -0.112,Y -342.983,Z 526.398,A 0.000,B 0.000,C 90.000,E1 71.692} C_DIS
LIN {X -0.035,Y -331.212,Z 526.379,A 0.000,B 0.000,C 90.000,E1 68.284} C_DIS
LIN {X -0.102,Y -321.330,Z 526.362,A 0.000,B 0.000,C 90.000,E1 65.153} C_DIS
LIN {X 0.102,Y -315.662,Z 526.351,A 0.000,B 0.000,C 90.000,E1 63.204} C_DIS
LIN {X -0.122,Y -308.025,Z 526.337,A 0.000,B 0.000,C 90.000,E1 60.667} C_DIS
LIN {X -0.065,Y -300.424,Z 526.322,A 0.000,B 0.000,C 90.000,E1 58.043} C_DIS
LIN {X 0.127,Y -291.364,Z 526.304,A 0.000,B 0.000,C 90.000,E1 54.689} C_DIS
LIN {X -0.044,Y -284.433,Z 526.289,A 0.000,B 0.000,C 90.000,E1 52.029} C_DIS
LIN {X -0.055,Y -278.983,Z 526.278,A 0.000,B 0.000,C 90.000,E1 49.989} C_DIS
LIN {X -0.023,Y -275.070,Z 526.270,A 0.000,B 0.000,C 90.000,E1 48.609} C_DIS
LIN {X -0.064,Y -268.657,Z 526.258,A 0.000,B 0.000,C 90.000,E1 46.539} C_DIS
LIN {X -0.067,Y -261.740,Z 526.247,A 0.000,B 0.000,C 90.000,E1 44.433} C_DIS
LIN {X 0.040,Y -252.357,Z 526.231,A 0.000,B 0.000,C 90.000,E1 41.553} C_DIS
LIN {X -0.069,Y -243.359,Z 526.215,A 0.000,B 0.000,C 90.000,E1 38.669} C_DIS
LIN {X -0.108,Y -235.085,Z 526.198,A 0.000,B 0.000,C 90.000,E1 35.724} C_DIS
LIN {X 0.082,Y -227.598,Z 526.182,A 0.000,B 0.000,C 90.000,E1 32.673} C_DIS
LIN {X -0.090,Y -220.883,Z 526.165,A 0.000,B 0.000,C 90.000,E1 29.667} C_DIS
LIN {X 0.042,Y -215.020,Z 526.148,A 0.000,B 0.000,C 90.000,E1 26.539} C_DIS
LIN {X 0.121,Y -209.971,Z 526.130,A 0.000,B 0.000,C 90.000,E1 23.387} C_DIS
LIN {X 0.028,Y -205.768,Z 526.113,A 0.000,B 0.000,C 90.000,E1 20.248} C_DIS
LIN {X 0.002,Y -201.493,Z 526.090,A 0.000,B 0.000,C 90.000,E1 16.260} C_DIS
LIN {X -0.006,Y -197.653,Z 526.063,A 0.000,B 0.000,C 90.000,E1 11.422} C_DIS
LIN {X -0.077,Y -194.898,Z 526.027,A 0.000,B 0.000,C 90.000,E1 4.935} C_DIS
LIN {X 0.055,Y -196.174,Z 525.966,A 0.000,B 0.000,C 90.000,E1 353.799} C_DIS
LIN {X 0.030,Y -199.710,Z 525.934,A 0.000,B 0.000,C 90.000,E1 348.117} C_DIS
LIN {X 0.075,Y -204.149,Z 525.907,A 0.000,B 0.000,C 90.000,E1 343.268} C_DIS
LIN {X 0.120,Y -208.791,Z 525.885,A 0.000,B 0.000,C 90.000,E1 339.263} C_DIS
LIN {X -0.049,Y -214.127,Z 525.863,A 0.000,B 0.000,C 90.000,E1 335.357} C_DIS
LIN {X 0.009,Y -220.072,Z 525.841,A 0.000,B 0.000,C 90.000,E1 331.435} C_DIS
LIN {X 0.000,Y -226.528,Z 525.820,A 0.000,B 0.000,C 90.000,E1 327.582} C_DIS
LIN {X -0.020,Y -233.701,Z 525.799,A 0.000,B 0.000,C 90.000,E1 323.783} C_DIS
LIN {X -0.008,Y -241.375,Z 525.778,A 0.000,B 0.000,C 90.000,E1 320.033} C_DIS
LIN {X 0.023,Y -250.029,Z 525.757,A 0.000,B 0.000,C 90.000,E1 316.338} C_DIS
LIN {X 0.144,Y -259.951,Z 525.737,A 0.000,B 0.000,C 90.000,E1 312.690} C_DIS
LIN {X -0.090,Y -271.061,Z 525.718,A 0.000,B 0.000,C 90.000,E1 309.197} C_DIS
LIN {X -0.067,Y -283.477,Z 525.698,A 0.000,B 0.000,C 90.000,E1 305.724} C_DIS
LIN {X -0.072,Y -297.212,Z 525.680,A 0.000,B 0.000,C 90.000,E1 302.339} C_DIS
LIN {X -0.003,Y -312.044,Z 525.661,A 0.000,B 0.000,C 90.000,E1 299.027} C_DIS
LIN {X 0.163,Y -326.579,Z 525.645,A 0.000,B 0.000,C 90.000,E1 296.104} C_DIS
LIN {X -0.067,Y -335.600,Z 525.636,A 0.000,B 0.000,C 90.000,E1 294.567} C_DIS
LIN {X 0.041,Y -351.377,Z 525.623,A 0.000,B 0.000,C 90.000,E1 292.078} C_DIS
LIN {X -0.035,Y -368.824,Z 525.609,A 0.000,B 0.000,C 90.000,E1 289.685} C_DIS
LIN {X 0.083,Y -387.775,Z 525.596,A 0.000,B 0.000,C 90.000,E1 287.330} C_DIS
LIN {X -0.113,Y -404.850,Z 525.585,A 0.000,B 0.000,C 90.000,E1 285.371} C_DIS
LIN {X -0.058,Y -419.754,Z 525.576,A 0.000,B 0.000,C 90.000,E1 283.703} C_DIS
LIN {X 0.142,Y -429.513,Z 525.570,A 0.000,B 0.000,C 90.000,E1 282.591} C_DIS
LIN {X 0.219,Y -441.175,Z 525.563,A 0.000,B 0.000,C 90.000,E1 281.243} C_DIS
LIN {X 0.150,Y -450.024,Z 525.557,A 0.000,B 0.000,C 90.000,E1 280.197} C_DIS
LIN {X 0.187,Y -458.116,Z 525.551,A 0.000,B 0.000,C 90.000,E1 279.151} C_DIS
LIN {X 0.035,Y -463.668,Z 525.547,A 0.000,B 0.000,C 90.000,E1 278.398} C_DIS
LIN {X -0.079,Y -468.676,Z 525.542,A 0.000,B 0.000,C 90.000,E1 277.644} C_DIS
LIN {X -0.146,Y -473.183,Z 525.538,A 0.000,B 0.000,C 90.000,E1 276.891} C_DIS
LIN {X -0.236,Y -477.233,Z 525.534,A 0.000,B 0.000,C 90.000,E1 276.144} C_DIS
LIN {X 0.241,Y -480.670,Z 525.530,A 0.000,B 0.000,C 90.000,E1 275.334} C_DIS
LIN {X 0.221,Y -483.416,Z 525.526,A 0.000,B 0.000,C 90.000,E1 274.588} C_DIS
LIN {X -0.127,Y -484.843,Z 525.523,A 0.000,B 0.000,C 90.000,E1 274.131} C_DIS
LIN {X 0.054,Y -485.951,Z 525.520,A 0.000,B 0.000,C 90.000,E1 273.612} C_DIS
LIN {X 0.239,Y -486.699,Z 525.517,A 0.000,B 0.000,C 90.000,E1 273.094} C_DIS
LIN {X -0.081,Y -487.166,Z 525.515,A 0.000,B 0.000,C 90.000,E1 272.636} C_DIS
LIN {X 0.091,Y -487.311,Z 525.512,A 0.000,B 0.000,C 90.000,E1 272.121} C_DIS
LIN {X -0.203,Y -487.036,Z 525.509,A 0.000,B 0.000,C 90.000,E1 271.661} C_DIS
LIN {X -0.026,Y -486.370,Z 525.506,A 0.000,B 0.000,C 90.000,E1 271.146} C_DIS
LIN {X 0.150,Y -485.270,Z 525.504,A 0.000,B 0.000,C 90.000,E1 270.630} C_DIS
LIN {X -0.161,Y -483.667,Z 525.501,A 0.000,B 0.000,C 90.000,E1 270.172} C_DIS
LIN {X 0.164,Y -482.675,Z 525.499,A 0.000,B 0.000,C 90.000,E1 269.885} C_DIS
LIN {X -0.159,Y -480.063,Z 525.497,A 0.000,B 0.000,C 90.000,E1 269.427} C_DIS
LIN {X 0.156,Y -478.526,Z 525.495,A 0.000,B 0.000,C 90.000,E1 269.141} C_DIS
LIN {X -0.016,Y -476.681,Z 525.494,A 0.000,B 0.000,C 90.000,E1 268.912} C_DIS
LIN {X 0.106,Y -472.256,Z 525.491,A 0.000,B 0.000,C 90.000,E1 268.396} C_DIS
LIN {X -0.059,Y -469.622,Z 525.490,A 0.000,B 0.000,C 90.000,E1 268.165} C_DIS
LIN {X 0.231,Y -463.642,Z 525.487,A 0.000,B 0.000,C 90.000,E1 267.650} C_DIS
LIN {X -0.055,Y -460.557,Z 525.486,A 0.000,B 0.000,C 90.000,E1 267.478} C_DIS
LIN {X 0.141,Y -453.773,Z 525.484,A 0.000,B 0.000,C 90.000,E1 267.078} C_DIS
LIN {X -0.008,Y -446.777,Z 525.482,A 0.000,B 0.000,C 90.000,E1 266.788} C_DIS
LIN {X -0.195,Y -439.695,Z 525.481,A 0.000,B 0.000,C 90.000,E1 266.560} C_DIS
LIN {X -0.056,Y -432.429,Z 525.480,A 0.000,B 0.000,C 90.000,E1 266.331} C_DIS
LIN {X -0.019,Y -424.368,Z 525.479,A 0.000,B 0.000,C 90.000,E1 266.159} C_DIS
LIN {X -0.027,Y -414.875,Z 525.478,A 0.000,B 0.000,C 90.000,E1 266.045} C_DIS
LIN {X 0.105,Y -407.759,Z 525.478,A 0.000,B 0.000,C 90.000,E1 265.988} C_DIS
LIN {X 0.027,Y -180.920,Z 525.478,A 0.000,B 0.000,C 90.000,E1 265.988} C_DIS
LIN {X 0.082,Y -180.857,Z 525.472,A 0.000,B 0.000,C 90.000,E1 264.951} C_DIS
LIN {X -0.019,Y -178.909,Z 525.443,A 0.000,B 0.000,C 90.000,E1 259.746} C_DIS
LIN {X 0.062,Y -175.952,Z 525.415,A 0.000,B 0.000,C 90.000,E1 254.629} C_DIS
LIN {X 0.008,Y -175.418,Z 525.410,A 0.000,B 0.000,C 90.000,E1 253.795} C_DIS
LIN {X 0.011,Y -172.181,Z 525.386,A 0.000,B 0.000,C 90.000,E1 249.518} C_DIS
LIN {X 0.050,Y -171.652,Z 525.381,A 0.000,B 0.000,C 90.000,E1 248.646} C_DIS
LIN {X 0.044,Y -167.876,Z 525.357,A 0.000,B 0.000,C 90.000,E1 244.332} C_DIS
LIN {X -0.012,Y -166.612,Z 525.348,A 0.000,B 0.000,C 90.000,E1 242.615} C_DIS
LIN {X -0.018,Y -162.599,Z 525.324,A 0.000,B 0.000,C 90.000,E1 238.250} C_DIS
LIN {X -0.044,Y -161.284,Z 525.314,A 0.000,B 0.000,C 90.000,E1 236.501} C_DIS
LIN {X -0.009,Y -157.283,Z 525.289,A 0.000,B 0.000,C 90.000,E1 232.065} C_DIS
LIN {X 0.013,Y -156.001,Z 525.279,A 0.000,B 0.000,C 90.000,E1 230.275} C_DIS
LIN {X -0.026,Y -152.259,Z 525.254,A 0.000,B 0.000,C 90.000,E1 225.810} C_DIS
LIN {X -0.004,Y -150.497,Z 525.239,A 0.000,B 0.000,C 90.000,E1 223.095} C_DIS
LIN {X 0.026,Y -147.221,Z 525.214,A 0.000,B 0.000,C 90.000,E1 218.543} C_DIS
LIN {X -0.004,Y -145.244,Z 525.194,A 0.000,B 0.000,C 90.000,E1 214.898} C_DIS
LIN {X -0.088,Y -142.362,Z 525.163,A 0.000,B 0.000,C 90.000,E1 209.411} C_DIS
LIN {X 0.033,Y -141.748,Z 525.153,A 0.000,B 0.000,C 90.000,E1 207.513} C_DIS
LIN {X -0.041,Y -139.492,Z 525.117,A 0.000,B 0.000,C 90.000,E1 201.046} C_DIS
LIN {X -0.004,Y -138.997,Z 525.101,A 0.000,B 0.000,C 90.000,E1 198.236} C_DIS
LIN {X -0.048,Y -138.337,Z 525.055,A 0.000,B 0.000,C 90.000,E1 189.849} C_DIS
LIN {X -0.025,Y -139.414,Z 525.008,A 0.000,B 0.000,C 90.000,E1 181.432} C_DIS
LIN {X 0.028,Y -141.327,Z 524.972,A 0.000,B 0.000,C 90.000,E1 174.894} C_DIS
LIN {X -0.015,Y -142.685,Z 524.956,A 0.000,B 0.000,C 90.000,E1 172.129} C_DIS
LIN {X -0.035,Y -145.044,Z 524.931,A 0.000,B 0.000,C 90.000,E1 167.521} C_DIS
LIN {X -0.038,Y -147.670,Z 524.910,A 0.000,B 0.000,C 90.000,E1 163.850} C_DIS
LIN {X -0.004,Y -150.312,Z 524.890,A 0.000,B 0.000,C 90.000,E1 160.188} C_DIS
LIN {X 0.008,Y -153.725,Z 524.870,A 0.000,B 0.000,C 90.000,E1 156.561} C_DIS
LIN {X -0.079,Y -157.138,Z 524.850,A 0.000,B 0.000,C 90.000,E1 152.999} C_DIS
LIN {X -0.005,Y -161.286,Z 524.830,A 0.000,B 0.000,C 90.000,E1 149.410} C_DIS
LIN {X 0.013,Y -164.403,Z 524.815,A 0.000,B 0.000,C 90.000,E1 146.755} C_DIS
LIN {X 0.010,Y -169.083,Z 524.796,A 0.000,B 0.000,C 90.000,E1 143.256} C_DIS
LIN {X -0.039,Y -171.640,Z 524.786,A 0.000,B 0.000,C 90.000,E1 141.537} C_DIS
LIN {X 0.008,Y -176.601,Z 524.767,A 0.000,B 0.000,C 90.000,E1 138.081} C_DIS
LIN {X 0.010,Y -180.900,Z 524.753,A 0.000,B 0.000,C 90.000,E1 135.526} C_DIS
LIN {X 0.001,Y -186.316,Z 524.734,A 0.000,B 0.000,C 90.000,E1 132.162} C_DIS
LIN {X 0.059,Y -191.420,Z 524.719,A 0.000,B 0.000,C 90.000,E1 129.358} C_DIS
LIN {X -0.006,Y -192.249,Z 524.716,A 0.000,B 0.000,C 90.000,E1 128.874} C_DIS
LIN {X -0.038,Y -289.576,Z 524.716,A 0.000,B 0.000,C 90.000,E1 128.874} C_DIS
LIN {X 0.040,Y -291.179,Z 524.716,A 0.000,B 0.000,C 90.000,E1 128.830} C_DIS
LIN {X -0.041,Y -294.475,Z 524.715,A 0.000,B 0.000,C 90.000,E1 128.705} C_DIS
LIN {X -0.173,Y -297.849,Z 524.714,A 0.000,B 0.000,C 90.000,E1 128.463} C_DIS
LIN {X -0.050,Y -301.508,Z 524.711,A 0.000,B 0.000,C 90.000,E1 127.971} C_DIS
LIN {X -0.106,Y -303.323,Z 524.709,A 0.000,B 0.000,C 90.000,E1 127.649} C_DIS
LIN {X 0.077,Y -304.741,Z 524.707,A 0.000,B 0.000,C 90.000,E1 127.282} C_DIS
LIN {X -0.132,Y -306.770,Z 524.704,A 0.000,B 0.000,C 90.000,E1 126.664} C_DIS
LIN {X 0.063,Y -316.742,Z 524.685,A 0.000,B 0.000,C 90.000,E1 123.372} C_DIS
LIN {X -0.026,Y -327.031,Z 524.669,A 0.000,B 0.000,C 90.000,E1 120.512} C_DIS
LIN {X -0.051,Y -338.672,Z 524.654,A 0.000,B 0.000,C 90.000,E1 117.692} C_DIS
LIN {X 0.106,Y -351.763,Z 524.638,A 0.000,B 0.000,C 90.000,E1 114.899} C_DIS
LIN {X -0.036,Y -364.718,Z 524.625,A 0.000,B 0.000,C 90.000,E1 112.514} C_DIS
LIN {X -0.148,Y -379.008,Z 524.612,A 0.000,B 0.000,C 90.000,E1 110.174} C_DIS
LIN {X -0.168,Y -394.738,Z 524.599,A 0.000,B 0.000,C 90.000,E1 107.873} C_DIS
LIN {X -0.026,Y -412.024,Z 524.587,A 0.000,B 0.000,C 90.000,E1 105.607} C_DIS
LIN {X 0.048,Y -430.985,Z 524.575,A 0.000,B 0.000,C 90.000,E1 103.411} C_DIS
LIN {X -0.052,Y -451.081,Z 524.563,A 0.000,B 0.000,C 90.000,E1 101.366} C_DIS
LIN {X -0.224,Y -471.730,Z 524.553,A 0.000,B 0.000,C 90.000,E1 99.500} C_DIS
LIN {X -0.028,Y -476.968,Z 524.550,A 0.000,B 0.000,C 90.000,E1 99.029} C_DIS
LIN {X 0.017,Y -479.187,Z 524.549,A 0.000,B 0.000,C 90.000,E1 98.803} C_DIS
LIN {X -0.066,Y -481.032,Z 524.548,A 0.000,B 0.000,C 90.000,E1 98.568} C_DIS
LIN {X -0.221,Y -482.428,Z 524.546,A 0.000,B 0.000,C 90.000,E1 98.341} C_DIS
LIN {X 0.015,Y -484.246,Z 524.543,A 0.000,B 0.000,C 90.000,E1 97.814} C_DIS
LIN {X 0.191,Y -484.965,Z 524.541,A 0.000,B 0.000,C 90.000,E1 97.296} C_DIS
LIN {X -0.102,Y -484.704,Z 524.538,A 0.000,B 0.000,C 90.000,E1 96.834} C_DIS
LIN {X 0.089,Y -483.424,Z 524.535,A 0.000,B 0.000,C 90.000,E1 96.315} C_DIS
LIN {X -0.082,Y -482.338,Z 524.534,A 0.000,B 0.000,C 90.000,E1 96.087} C_DIS
LIN {X -0.201,Y -480.878,Z 524.532,A 0.000,B 0.000,C 90.000,E1 95.853} C_DIS
LIN {X -0.065,Y -470.932,Z 524.525,A 0.000,B 0.000,C 90.000,E1 94.588} C_DIS
LIN {X 0.173,Y -459.390,Z 524.517,A 0.000,B 0.000,C 90.000,E1 93.037} C_DIS
LIN {X -0.025,Y -450.600,Z 524.510,A 0.000,B 0.000,C 90.000,E1 91.776} C_DIS
LIN {X 0.196,Y -437.973,Z 524.498,A 0.000,B 0.000,C 90.000,E1 89.656} C_DIS
LIN {X -0.007,Y -426.677,Z 524.488,A 0.000,B 0.000,C 90.000,E1 87.822} C_DIS
LIN {X -0.212,Y -412.324,Z 524.474,A 0.000,B 0.000,C 90.000,E1 85.412} C_DIS
LIN {X 0.038,Y -399.760,Z 524.462,A 0.000,B 0.000,C 90.000,E1 83.166} C_DIS
LIN {X -0.024,Y -390.418,Z 524.453,A 0.000,B 0.000,C 90.000,E1 81.489} C_DIS
LIN {X -0.159,Y -379.493,Z 524.442,A 0.000,B 0.000,C 90.000,E1 79.511} C_DIS
LIN {X -0.046,Y -362.642,Z 524.424,A 0.000,B 0.000,C 90.000,E1 76.284} C_DIS
LIN {X -0.148,Y -353.097,Z 524.412,A 0.000,B 0.000,C 90.000,E1 74.212} C_DIS
LIN {X 0.084,Y -344.482,Z 524.400,A 0.000,B 0.000,C 90.000,E1 72.054} C_DIS
LIN {X 0.093,Y -333.614,Z 524.383,A 0.000,B 0.000,C 90.000,E1 68.975} C_DIS
LIN {X -0.048,Y -323.564,Z 524.366,A 0.000,B 0.000,C 90.000,E1 65.869} C_DIS
LIN {X -0.084,Y -315.924,Z 524.352,A 0.000,B 0.000,C 90.000,E1 63.332} C_DIS
LIN {X 0.122,Y -308.273,Z 524.337,A 0.000,B 0.000,C 90.000,E1 60.717} C_DIS
LIN {X 0.028,Y -300.664,Z 524.323,A 0.000,B 0.000,C 90.000,E1 58.122} C_DIS
LIN {X -0.020,Y -291.546,Z 524.305,A 0.000,B 0.000,C 90.000,E1 54.815} C_DIS
LIN {X 0.046,Y -284.610,Z 524.290,A 0.000,B 0.000,C 90.000,E1 52.110} C_DIS
LIN {X 0.037,Y -279.165,Z 524.278,A 0.000,B 0.000,C 90.000,E1 50.070} C_DIS
LIN {X 0.069,Y -275.286,Z 524.271,A 0.000,B 0.000,C 90.000,E1 48.690} C_DIS
LIN {X 0.028,Y -268.894,Z 524.259,A 0.000,B 0.000,C 90.000,E1 46.620} C_DIS
LIN {X 0.028,Y -261.980,Z 524.247,A 0.000,B 0.000,C 90.000,E1 44.514} C_DIS
LIN {X -0.051,Y -252.607,Z 524.231,A 0.000,B 0.000,C 90.000,E1 41.676} C_DIS
LIN {X 0.033,Y -243.585,Z 524.215,A 0.000,B 0.000,C 90.000,E1 38.749} C_DIS
LIN {X -0.008,Y -235.291,Z 524.199,A 0.000,B 0.000,C 90.000,E1 35.804} C_DIS
LIN {X -0.006,Y -227.795,Z 524.182,A 0.000,B 0.000,C 90.000,E1 32.801} C_DIS
LIN {X 0.021,Y -221.051,Z 524.165,A 0.000,B 0.000,C 90.000,E1 29.745} C_DIS
LIN {X -0.035,Y -215.159,Z 524.148,A 0.000,B 0.000,C 90.000,E1 26.668} C_DIS
LIN {X 0.050,Y -210.080,Z 524.131,A 0.000,B 0.000,C 90.000,E1 23.515} C_DIS
LIN {X -0.026,Y -204.922,Z 524.109,A 0.000,B 0.000,C 90.000,E1 19.577} C_DIS
LIN {X 0.055,Y -200.818,Z 524.086,A 0.000,B 0.000,C 90.000,E1 15.552} C_DIS
LIN {X 0.020,Y -197.189,Z 524.060,A 0.000,B 0.000,C 90.000,E1 10.715} C_DIS
LIN {X 0.065,Y -194.723,Z 524.023,A 0.000,B 0.000,C 90.000,E1 4.188} C_DIS
LIN {X 0.052,Y -196.091,Z 523.966,A 0.000,B 0.000,C 90.000,E1 353.799} C_DIS
LIN {X 0.024,Y -199.602,Z 523.934,A 0.000,B 0.000,C 90.000,E1 348.117} C_DIS
LIN {X -0.046,Y -203.208,Z 523.912,A 0.000,B 0.000,C 90.000,E1 344.102} C_DIS
LIN {X 0.096,Y -207.689,Z 523.889,A 0.000,B 0.000,C 90.000,E1 340.061} C_DIS
LIN {X 0.089,Y -212.886,Z 523.867,A 0.000,B 0.000,C 90.000,E1 336.102} C_DIS
LIN {X -0.083,Y -218.721,Z 523.846,A 0.000,B 0.000,C 90.000,E1 332.231} C_DIS
LIN {X 0.052,Y -225.097,Z 523.824,A 0.000,B 0.000,C 90.000,E1 328.329} C_DIS
LIN {X -0.009,Y -232.132,Z 523.803,A 0.000,B 0.000,C 90.000,E1 324.529} C_DIS
LIN {X -0.149,Y -239.674,Z 523.782,A 0.000,B 0.000,C 90.000,E1 320.803} C_DIS
LIN {X -0.001,Y -248.159,Z 523.761,A 0.000,B 0.000,C 90.000,E1 317.067} C_DIS
LIN {X 0.030,Y -256.800,Z 523.743,A 0.000,B 0.000,C 90.000,E1 313.785} C_DIS
LIN {X 0.037,Y -267.551,Z 523.723,A 0.000,B 0.000,C 90.000,E1 310.216} C_DIS
LIN {X -0.052,Y -279.605,Z 523.704,A 0.000,B 0.000,C 90.000,E1 306.744} C_DIS
LIN {X 0.154,Y -292.960,Z 523.685,A 0.000,B 0.000,C 90.000,E1 303.293} C_DIS
LIN {X -0.047,Y -305.956,Z 523.668,A 0.000,B 0.000,C 90.000,E1 300.335} C_DIS
LIN {X 0.007,Y -321.562,Z 523.650,A 0.000,B 0.000,C 90.000,E1 297.078} C_DIS
LIN {X 0.151,Y -330.074,Z 523.642,A 0.000,B 0.000,C 90.000,E1 295.463} C_DIS
LIN {X -0.048,Y -347.298,Z 523.626,A 0.000,B 0.000,C 90.000,E1 292.695} C_DIS
LIN {X -0.003,Y -359.919,Z 523.616,A 0.000,B 0.000,C 90.000,E1 290.865} C_DIS
LIN {X 0.044,Y -375.823,Z 523.604,A 0.000,B 0.000,C 90.000,E1 288.779} C_DIS
LIN {X 0.187,Y -392.652,Z 523.593,A 0.000,B 0.000,C 90.000,E1 286.732} C_DIS
LIN {X -0.200,Y -412.390,Z 523.581,A 0.000,B 0.000,C 90.000,E1 284.537} C_DIS
LIN {X -0.138,Y -427.249,Z 523.571,A 0.000,B 0.000,C 90.000,E1 282.883} C_DIS
LIN {X -0.029,Y -438.947,Z 523.564,A 0.000,B 0.000,C 90.000,E1 281.535} C_DIS
LIN {X -0.131,Y -448.012,Z 523.558,A 0.000,B 0.000,C 90.000,E1 280.489} C_DIS
LIN {X -0.123,Y -456.306,Z 523.552,A 0.000,B 0.000,C 90.000,E1 279.443} C_DIS
LIN {X 0.228,Y -462.015,Z 523.548,A 0.000,B 0.000,C 90.000,E1 278.624} C_DIS
LIN {X 0.105,Y -467.211,Z 523.544,A 0.000,B 0.000,C 90.000,E1 277.871} C_DIS
LIN {X -0.040,Y -471.901,Z 523.540,A 0.000,B 0.000,C 90.000,E1 277.125} C_DIS
LIN {X 0.192,Y -477.375,Z 523.534,A 0.000,B 0.000,C 90.000,E1 276.087} C_DIS
LIN {X 0.195,Y -480.817,Z 523.530,A 0.000,B 0.000,C 90.000,E1 275.334} C_DIS
LIN {X 0.177,Y -483.581,Z 523.526,A 0.000,B 0.000,C 90.000,E1 274.588} C_DIS
LIN {X -0.170,Y -485.009,Z 523.523,A 0.000,B 0.000,C 90.000,E1 274.131} C_DIS
LIN {X 0.011,Y -486.092,Z 523.520,A 0.000,B 0.000,C 90.000,E1 273.612} C_DIS
LIN {X 0.198,Y -486.845,Z 523.517,A 0.000,B 0.000,C 90.000,E1 273.094} C_DIS
LIN {X -0.122,Y -487.295,Z 523.515,A 0.000,B 0.000,C 90.000,E1 272.636} C_DIS
LIN {X 0.051,Y -487.409,Z 523.512,A 0.000,B 0.000,C 90.000,E1 272.121} C_DIS
LIN {X 0.244,Y -487.147,Z 523.509,A 0.000,B 0.000,C 90.000,E1 271.604} C_DIS
LIN {X -0.065,Y -486.489,Z 523.506,A 0.000,B 0.000,C 90.000,E1 271.146} C_DIS
LIN {X 0.113,Y -485.340,Z 523.504,A 0.000,B 0.000,C 90.000,E1 270.630} C_DIS
LIN {X -0.198,Y -483.733,Z 523.501,A 0.000,B 0.000,C 90.000,E1 270.172} C_DIS
LIN {X -0.031,Y -481.492,Z 523.498,A 0.000,B 0.000,C 90.000,E1 269.656} C_DIS
LIN {X 0.120,Y -478.523,Z 523.495,A 0.000,B 0.000,C 90.000,E1 269.141} C_DIS
LIN {X -0.222,Y -474.605,Z 523.493,A 0.000,B 0.000,C 90.000,E1 268.682} C_DIS
LIN {X -0.094,Y -469.638,Z 523.490,A 0.000,B 0.000,C 90.000,E1 268.165} C_DIS
LIN {X 0.151,Y -463.509,Z 523.487,A 0.000,B 0.000,C 90.000,E1 267.650} C_DIS
LIN {X 0.064,Y -456.934,Z 523.485,A 0.000,B 0.000,C 90.000,E1 267.249} C_DIS
LIN {X 0.074,Y -449.847,Z 523.483,A 0.000,B 0.000,C 90.000,E1 266.906} C_DIS
LIN {X 0.199,Y -442.931,Z 523.481,A 0.000,B 0.000,C 90.000,E1 266.617} C_DIS
LIN {X 0.164,Y -435.685,Z 523.480,A 0.000,B 0.000,C 90.000,E1 266.388} C_DIS
LIN {X 0.015,Y -427.741,Z 523.479,A 0.000,B 0.000,C 90.000,E1 266.216} C_DIS
LIN {X -0.155,Y -419.222,Z 523.478,A 0.000,B 0.000,C 90.000,E1 266.102} C_DIS
LIN {X 0.159,Y -410.694,Z 523.478,A 0.000,B 0.000,C 90.000,E1 265.988} C_DIS
LIN {X 0.065,Y -405.587,Z 523.478,A 0.000,B 0.000,C 90.000,E1 265.988} C_DIS
LIN {X 0.009,Y -180.920,Z 523.478,A 0.000,B 0.000,C 90.000,E1 265.988} C_DIS
LIN {X 0.064,Y -180.855,Z 523.472,A 0.000,B 0.000,C 90.000,E1 264.951} C_DIS
LIN {X -0.035,Y -178.906,Z 523.443,A 0.000,B 0.000,C 90.000,E1 259.746} C_DIS
LIN {X 0.044,Y -175.950,Z 523.415,A 0.000,B 0.000,C 90.000,E1 254.629} C_DIS
LIN {X -0.009,Y -175.414,Z 523.410,A 0.000,B 0.000,C 90.000,E1 253.795} C_DIS
LIN {X -0.006,Y -172.177,Z 523.386,A 0.000,B 0.000,C 90.000,E1 249.518} C_DIS
LIN {X 0.033,Y -171.648,Z 523.381,A 0.000,B 0.000,C 90.000,E1 248.646} C_DIS
LIN {X 0.028,Y -167.871,Z 523.357,A 0.000,B 0.000,C 90.000,E1 244.332} C_DIS
LIN {X -0.029,Y -166.606,Z 523.348,A 0.000,B 0.000,C 90.000,E1 242.615} C_DIS
LIN {X -0.035,Y -162.595,Z 523.324,A 0.000,B 0.000,C 90.000,E1 238.250} C_DIS
LIN {X -0.060,Y -161.279,Z 523.314,A 0.000,B 0.000,C 90.000,E1 236.501} C_DIS
LIN {X -0.025,Y -157.278,Z 523.289,A 0.000,B 0.000,C 90.000,E1 232.065} C_DIS
LIN {X -0.003,Y -155.997,Z 523.279,A 0.000,B 0.000,C 90.000,E1 230.275} C_DIS
LIN {X -0.042,Y -152.255,Z 523.254,A 0.000,B 0.000,C 90.000,E1 225.810} C_DIS
LIN {X -0.020,Y -150.493,Z 523.239,A 0.000,B 0.000,C 90.000,E1 223.095} C_DIS
LIN {X 0.010,Y -147.218,Z 523.214,A 0.000,B 0.000,C 90.000,E1 218.543} C_DIS
LIN {X -0.020,Y -145.239,Z 523.194,A 0.000,B 0.000,C 90.000,E1 214.898} C_DIS
LIN {X 0.021,Y -142.360,Z 523.163,A 0.000,B 0.000,C 90.000,E1 209.361} C_DIS
LIN {X 0.018,Y -141.746,Z 523.153,A 0.000,B 0.000,C 90.000,E1 207.513} C_DIS
LIN {X -0.056,Y -139.491,Z 523.117,A 0.000,B 0.000,C 90.000,E1 201.046} C_DIS
LIN {X -0.019,Y -138.995,Z 523.101,A 0.000,B 0.000,C 90.000,E1 198.236} C_DIS
LIN {X -0.063,Y -138.336,Z 523.055,A 0.000,B 0.000,C 90.000,E1 189.849} C_DIS
LIN {X -0.040,Y -139.416,Z 523.008,A 0.000,B 0.000,C 90.000,E1 181.432} C_DIS
LIN {X 0.013,Y -141.330,Z 522.972,A 0.000,B 0.000,C 90.000,E1 174.894} C_DIS
LIN {X -0.030,Y -142.687,Z 522.956,A 0.000,B 0.000,C 90.000,E1 172.129} C_DIS
LIN {X -0.051,Y -145.048,Z 522.931,A 0.000,B 0.000,C 90.000,E1 167.521} C_DIS
LIN {X 0.088,Y -147.674,Z 522.910,A 0.000,B 0.000,C 90.000,E1 163.795} C_DIS
LIN {X -0.019,Y -150.317,Z 522.890,A 0.000,B 0.000,C 90.000,E1 160.188} C_DIS
LIN {X 0.053,Y -153.731,Z 522.870,A 0.000,B 0.000,C 90.000,E1 156.538} C_DIS
LIN {X 0.044,Y -157.145,Z 522.850,A 0.000,B 0.000,C 90.000,E1 152.948} C_DIS
LIN {X -0.021,Y -161.293,Z 522.830,A 0.000,B 0.000,C 90.000,E1 149.410} C_DIS
LIN {X -0.003,Y -164.410,Z 522.815,A 0.000,B 0.000,C 90.000,E1 146.755} C_DIS
LIN {X -0.007,Y -169.091,Z 522.796,A 0.000,B 0.000,C 90.000,E1 143.256} C_DIS
LIN {X -0.056,Y -171.647,Z 522.786,A 0.000,B 0.000,C 90.000,E1 141.537} C_DIS
LIN {X -0.010,Y -176.610,Z 522.767,A 0.000,B 0.000,C 90.000,E1 138.081} C_DIS
LIN {X -0.008,Y -180.909,Z 522.753,A 0.000,B 0.000,C 90.000,E1 135.526} C_DIS
LIN {X -0.017,Y -186.325,Z 522.734,A 0.000,B 0.000,C 90.000,E1 132.162} C_DIS
LIN {X 0.039,Y -191.429,Z 522.719,A 0.000,B 0.000,C 90.000,E1 129.358} C_DIS
LIN {X 0.104,Y -192.268,Z 522.716,A 0.000,B 0.000,C 90.000,E1 128.830} C_DIS
LIN {X 0.128,Y -289.537,Z 522.716,A 0.000,B 0.000,C 90.000,E1 128.830} C_DIS
LIN {X 0.011,Y -290.911,Z 522.716,A 0.000,B 0.000,C 90.000,E1 128.830} C_DIS
LIN {X 0.026,Y -294.044,Z 522.715,A 0.000,B 0.000,C 90.000,E1 128.705} C_DIS
LIN {X 0.009,Y -297.371,Z 522.714,A 0.000,B 0.000,C 90.000,E1 128.463} C_DIS
LIN {X 0.043,Y -301.036,Z 522.711,A 0.000,B 0.000,C 90.000,E1 128.016} C_DIS
LIN {X -0.164,Y -302.930,Z 522.709,A 0.000,B 0.000,C 90.000,E1 127.729} C_DIS
LIN {X 0.053,Y -304.410,Z 522.708,A 0.000,B 0.000,C 90.000,E1 127.363} C_DIS
LIN {X 0.069,Y -305.589,Z 522.706,A 0.000,B 0.000,C 90.000,E1 127.030} C_DIS
LIN {X 0.032,Y -316.477,Z 522.686,A 0.000,B 0.000,C 90.000,E1 123.452} C_DIS
LIN {X -0.059,Y -326.732,Z 522.670,A 0.000,B 0.000,C 90.000,E1 120.590} C_DIS
LIN {X -0.089,Y -338.337,Z 522.654,A 0.000,B 0.000,C 90.000,E1 117.769} C_DIS
LIN {X 0.064,Y -351.390,Z 522.639,A 0.000,B 0.000,C 90.000,E1 114.975} C_DIS
LIN {X -0.081,Y -364.307,Z 522.625,A 0.000,B 0.000,C 90.000,E1 112.589} C_DIS
LIN {X -0.196,Y -378.558,Z 522.612,A 0.000,B 0.000,C 90.000,E1 110.248} C_DIS
LIN {X -0.099,Y -394.245,Z 522.600,A 0.000,B 0.000,C 90.000,E1 107.928} C_DIS
LIN {X 0.028,Y -411.485,Z 522.587,A 0.000,B 0.000,C 90.000,E1 105.662} C_DIS
LIN {X -0.015,Y -430.400,Z 522.575,A 0.000,B 0.000,C 90.000,E1 103.480} C_DIS
LIN {X -0.059,Y -450.480,Z 522.563,A 0.000,B 0.000,C 90.000,E1 101.422} C_DIS
LIN {X 0.193,Y -471.114,Z 522.553,A 0.000,B 0.000,C 90.000,E1 99.500} C_DIS
LIN {X -0.160,Y -476.350,Z 522.550,A 0.000,B 0.000,C 90.000,E1 99.095} C_DIS
LIN {X -0.046,Y -478.763,Z 522.549,A 0.000,B 0.000,C 90.000,E1 98.859} C_DIS
LIN {X -0.030,Y -480.676,Z 522.548,A 0.000,B 0.000,C 90.000,E1 98.624} C_DIS
LIN {X -0.086,Y -482.138,Z 522.547,A 0.000,B 0.000,C 90.000,E1 98.398} C_DIS
LIN {X -0.208,Y -483.323,Z 522.545,A 0.000,B 0.000,C 90.000,E1 98.163} C_DIS
LIN {X 0.147,Y -484.187,Z 522.544,A 0.000,B 0.000,C 90.000,E1 97.871} C_DIS
LIN {X -0.153,Y -485.091,Z 522.541,A 0.000,B 0.000,C 90.000,E1 97.409} C_DIS
LIN {X 0.033,Y -485.008,Z 522.538,A 0.000,B 0.000,C 90.000,E1 96.891} C_DIS
LIN {X 0.225,Y -483.925,Z 522.536,A 0.000,B 0.000,C 90.000,E1 96.372} C_DIS
LIN {X 0.055,Y -482.957,Z 522.534,A 0.000,B 0.000,C 90.000,E1 96.144} C_DIS
LIN {X -0.064,Y -481.643,Z 522.533,A 0.000,B 0.000,C 90.000,E1 95.910} C_DIS
LIN {X 0.112,Y -477.886,Z 522.530,A 0.000,B 0.000,C 90.000,E1 95.391} C_DIS
LIN {X 0.056,Y -462.035,Z 522.519,A 0.000,B 0.000,C 90.000,E1 93.383} C_DIS
LIN {X 0.124,Y -451.315,Z 522.510,A 0.000,B 0.000,C 90.000,E1 91.835} C_DIS
LIN {X 0.102,Y -437.000,Z 522.497,A 0.000,B 0.000,C 90.000,E1 89.484} C_DIS
LIN {X -0.113,Y -425.672,Z 522.487,A 0.000,B 0.000,C 90.000,E1 87.650} C_DIS
LIN {X -0.019,Y -412.915,Z 522.475,A 0.000,B 0.000,C 90.000,E1 85.469} C_DIS
LIN {X -0.157,Y -400.346,Z 522.463,A 0.000,B 0.000,C 90.000,E1 83.280} C_DIS
LIN {X -0.144,Y -389.417,Z 522.452,A 0.000,B 0.000,C 90.000,E1 81.310} C_DIS
LIN {X 0.018,Y -378.485,Z 522.440,A 0.000,B 0.000,C 90.000,E1 79.285} C_DIS
LIN {X 0.118,Y -364.608,Z 522.426,A 0.000,B 0.000,C 90.000,E1 76.645} C_DIS
LIN {X -0.007,Y -353.529,Z 522.413,A 0.000,B 0.000,C 90.000,E1 74.283} C_DIS
LIN {X -0.091,Y -343.738,Z 522.399,A 0.000,B 0.000,C 90.000,E1 71.873} C_DIS
LIN {X 0.005,Y -331.891,Z 522.380,A 0.000,B 0.000,C 90.000,E1 68.465} C_DIS
LIN {X -0.173,Y -321.947,Z 522.363,A 0.000,B 0.000,C 90.000,E1 65.357} C_DIS
LIN {X -0.100,Y -314.285,Z 522.349,A 0.000,B 0.000,C 90.000,E1 62.794} C_DIS
LIN {X -0.077,Y -306.628,Z 522.334,A 0.000,B 0.000,C 90.000,E1 60.205} C_DIS
LIN {X -0.056,Y -299.040,Z 522.320,A 0.000,B 0.000,C 90.000,E1 57.582} C_DIS
LIN {X -0.155,Y -289.998,Z 522.301,A 0.000,B 0.000,C 90.000,E1 54.276} C_DIS
LIN {X 0.165,Y -284.788,Z 522.290,A 0.000,B 0.000,C 90.000,E1 52.190} C_DIS
LIN {X -0.059,Y -279.370,Z 522.279,A 0.000,B 0.000,C 90.000,E1 50.194} C_DIS
LIN {X 0.006,Y -275.508,Z 522.271,A 0.000,B 0.000,C 90.000,E1 48.809} C_DIS
LIN {X -0.048,Y -269.130,Z 522.260,A 0.000,B 0.000,C 90.000,E1 46.743} C_DIS
LIN {X 0.148,Y -262.224,Z 522.248,A 0.000,B 0.000,C 90.000,E1 44.595} C_DIS
LIN {X 0.072,Y -252.874,Z 522.232,A 0.000,B 0.000,C 90.000,E1 41.757} C_DIS
LIN {X -0.029,Y -243.838,Z 522.216,A 0.000,B 0.000,C 90.000,E1 38.874} C_DIS
LIN {X -0.068,Y -235.531,Z 522.200,A 0.000,B 0.000,C 90.000,E1 35.931} C_DIS
LIN {X 0.131,Y -228.006,Z 522.183,A 0.000,B 0.000,C 90.000,E1 32.880} C_DIS
LIN {X -0.031,Y -221.237,Z 522.166,A 0.000,B 0.000,C 90.000,E1 29.873} C_DIS
LIN {X 0.112,Y -215.313,Z 522.149,A 0.000,B 0.000,C 90.000,E1 26.744} C_DIS
LIN {X 0.010,Y -210.204,Z 522.131,A 0.000,B 0.000,C 90.000,E1 23.643} C_DIS
LIN {X 0.009,Y -205.017,Z 522.109,A 0.000,B 0.000,C 90.000,E1 19.685} C_DIS
LIN {X 0.084,Y -200.889,Z 522.087,A 0.000,B 0.000,C 90.000,E1 15.662} C_DIS
LIN {X 0.008,Y -197.229,Z 522.060,A 0.000,B 0.000,C 90.000,E1 10.838} C_DIS
LIN {X 0.083,Y -194.701,Z 522.024,A 0.000,B 0.000,C 90.000,E1 4.302} C_DIS
LIN {X 0.049,Y -196.008,Z 521.966,A 0.000,B 0.000,C 90.000,E1 353.799} C_DIS
LIN {X 0.022,Y -198.874,Z 521.939,A 0.000,B 0.000,C 90.000,E1 348.926} C_DIS
LIN {X -0.057,Y -203.101,Z 521.912,A 0.000,B 0.000,C 90.000,E1 344.102} C_DIS
LIN {X 0.081,Y -207.560,Z 521.889,A 0.000,B 0.000,C 90.000,E1 340.061} C_DIS
LIN {X 0.070,Y -212.764,Z 521.867,A 0.000,B 0.000,C 90.000,E1 336.102} C_DIS
LIN {X -0.106,Y -218.611,Z 521.846,A 0.000,B 0.000,C 90.000,E1 332.231} C_DIS
LIN {X 0.024,Y -224.977,Z 521.824,A 0.000,B 0.000,C 90.000,E1 328.329} C_DIS
LIN {X 0.065,Y -230.612,Z 521.807,A 0.000,B 0.000,C 90.000,E1 325.261} C_DIS
LIN {X -0.127,Y -238.011,Z 521.786,A 0.000,B 0.000,C 90.000,E1 321.537} C_DIS
LIN {X -0.011,Y -246.327,Z 521.766,A 0.000,B 0.000,C 90.000,E1 317.796} C_DIS
LIN {X 0.152,Y -255.733,Z 521.745,A 0.000,B 0.000,C 90.000,E1 314.109} C_DIS
LIN {X 0.137,Y -266.384,Z 521.725,A 0.000,B 0.000,C 90.000,E1 310.539} C_DIS
LIN {X -0.032,Y -278.327,Z 521.706,A 0.000,B 0.000,C 90.000,E1 307.076} C_DIS
LIN {X -0.035,Y -291.569,Z 521.687,A 0.000,B 0.000,C 90.000,E1 303.658} C_DIS
LIN {X -0.115,Y -304.451,Z 521.670,A 0.000,B 0.000,C 90.000,E1 300.669} C_DIS
LIN {X 0.036,Y -319.923,Z 521.652,A 0.000,B 0.000,C 90.000,E1 297.385} C_DIS
LIN {X 0.099,Y -330.082,Z 521.642,A 0.000,B 0.000,C 90.000,E1 295.463} C_DIS
LIN {X -0.100,Y -347.292,Z 521.626,A 0.000,B 0.000,C 90.000,E1 292.695} C_DIS
LIN {X -0.002,Y -362.127,Z 521.614,A 0.000,B 0.000,C 90.000,E1 290.556} C_DIS
LIN {X -0.014,Y -375.825,Z 521.604,A 0.000,B 0.000,C 90.000,E1 288.779} C_DIS
LIN {X 0.128,Y -392.664,Z 521.593,A 0.000,B 0.000,C 90.000,E1 286.732} C_DIS
LIN {X -0.185,Y -412.335,Z 521.581,A 0.000,B 0.000,C 90.000,E1 284.537} C_DIS
LIN {X -0.124,Y -427.237,Z 521.571,A 0.000,B 0.000,C 90.000,E1 282.883} C_DIS
LIN {X -0.082,Y -439.041,Z 521.564,A 0.000,B 0.000,C 90.000,E1 281.535} C_DIS
LIN {X -0.185,Y -448.129,Z 521.558,A 0.000,B 0.000,C 90.000,E1 280.489} C_DIS
LIN {X -0.100,Y -456.470,Z 521.552,A 0.000,B 0.000,C 90.000,E1 279.434} C_DIS
LIN {X 0.176,Y -462.175,Z 521.548,A 0.000,B 0.000,C 90.000,E1 278.624} C_DIS
LIN {X 0.054,Y -467.372,Z 521.544,A 0.000,B 0.000,C 90.000,E1 277.871} C_DIS
LIN {X -0.090,Y -472.056,Z 521.540,A 0.000,B 0.000,C 90.000,E1 277.125} C_DIS
LIN {X 0.144,Y -477.507,Z 521.534,A 0.000,B 0.000,C 90.000,E1 276.087} C_DIS
LIN {X 0.148,Y -480.966,Z 521.530,A 0.000,B 0.000,C 90.000,E1 275.334} C_DIS
LIN {X 0.131,Y -483.709,Z 521.526,A 0.000,B 0.000,C 90.000,E1 274.588} C_DIS
LIN {X -0.216,Y -485.135,Z 521.523,A 0.000,B 0.000,C 90.000,E1 274.131} C_DIS
LIN {X -0.034,Y -486.236,Z 521.520,A 0.000,B 0.000,C 90.000,E1 273.612} C_DIS
LIN {X 0.153,Y -486.994,Z 521.517,A 0.000,B 0.000,C 90.000,E1 273.094} C_DIS
LIN {X -0.166,Y -487.426,Z 521.515,A 0.000,B 0.000,C 90.000,E1 272.636} C_DIS
LIN {X 0.008,Y -487.531,Z 521.512,A 0.000,B 0.000,C 90.000,E1 272.121} C_DIS
LIN {X 0.202,Y -487.263,Z 521.509,A 0.000,B 0.000,C 90.000,E1 271.604} C_DIS
LIN {X -0.107,Y -486.578,Z 521.506,A 0.000,B 0.000,C 90.000,E1 271.146} C_DIS
LIN {X 0.071,Y -485.474,Z 521.504,A 0.000,B 0.000,C 90.000,E1 270.630} C_DIS
LIN {X -0.238,Y -483.796,Z 521.501,A 0.000,B 0.000,C 90.000,E1 270.172} C_DIS
LIN {X -0.070,Y -481.484,Z 521.498,A 0.000,B 0.000,C 90.000,E1 269.656} C_DIS
LIN {X -0.234,Y -480.121,Z 521.497,A 0.000,B 0.000,C 90.000,E1 269.427} C_DIS
LIN {X -0.091,Y -476.688,Z 521.494,A 0.000,B 0.000,C 90.000,E1 268.912} C_DIS
LIN {X 0.213,Y -474.609,Z 521.492,A 0.000,B 0.000,C 90.000,E1 268.625} C_DIS
LIN {X -0.133,Y -469.601,Z 521.490,A 0.000,B 0.000,C 90.000,E1 268.165} C_DIS
LIN {X 0.157,Y -463.601,Z 521.487,A 0.000,B 0.000,C 90.000,E1 267.650} C_DIS
LIN {X 0.057,Y -456.934,Z 521.485,A 0.000,B 0.000,C 90.000,E1 267.249} C_DIS
LIN {X 0.095,Y -449.883,Z 521.483,A 0.000,B 0.000,C 90.000,E1 266.906} C_DIS
LIN {X -0.195,Y -443.188,Z 521.481,A 0.000,B 0.000,C 90.000,E1 266.674} C_DIS
LIN {X 0.175,Y -435.779,Z 521.480,A 0.000,B 0.000,C 90.000,E1 266.388} C_DIS
LIN {X 0.033,Y -428.113,Z 521.479,A 0.000,B 0.000,C 90.000,E1 266.216} C_DIS
LIN {X -0.175,Y -419.190,Z 521.478,A 0.000,B 0.000,C 90.000,E1 266.102} C_DIS
LIN {X 0.145,Y -410.932,Z 521.478,A 0.000,B 0.000,C 90.000,E1 265.988} C_DIS
LIN {X 0.054,Y -406.318,Z 521.478,A 0.000,B 0.000,C 90.000,E1 265.988} C_DIS
LIN {X 0.004,Y -180.919,Z 521.478,A 0.000,B 0.000,C 90.000,E1 265.988} C_DIS
LIN {X 0.060,Y -180.854,Z 521.472,A 0.000,B 0.000,C 90.000,E1 264.951} C_DIS
LIN {X -0.041,Y -178.905,Z 521.443,A 0.000,B 0.000,C 90.000,E1 259.746} C_DIS
LIN {X 0.040,Y -175.949,Z 521.415,A 0.000,B 0.000,C 90.000,E1 254.629} C_DIS
LIN {X -0.013,Y -175.412,Z 521.410,A 0.000,B 0.000,C 90.000,E1 253.795} C_DIS
LIN {X -0.010,Y -172.176,Z 521.386,A 0.000,B 0.000,C 90.000,E1 249.518} C_DIS
LIN {X 0.029,Y -171.647,Z 521.381,A 0.000,B 0.000,C 90.000,E1 248.646} C_DIS
LIN {X 0.024,Y -167.870,Z 521.357,A 0.000,B 0.000,C 90.000,E1 244.332} C_DIS
LIN {X -0.033,Y -166.605,Z 521.348,A 0.000,B 0.000,C 90.000,E1 242.615} C_DIS
LIN {X -0.039,Y -162.594,Z 521.324,A 0.000,B 0.000,C 90.000,E1 238.250} C_DIS
LIN {X -0.065,Y -161.278,Z 521.314,A 0.000,B 0.000,C 90.000,E1 236.501} C_DIS
LIN {X -0.030,Y -157.277,Z 521.289,A 0.000,B 0.000,C 90.000,E1 232.065} C_DIS
LIN {X -0.006,Y -155.996,Z 521.279,A 0.000,B 0.000,C 90.000,E1 230.275} C_DIS
LIN {X -0.046,Y -152.253,Z 521.254,A 0.000,B 0.000,C 90.000,E1 225.810} C_DIS
LIN {X -0.023,Y -150.493,Z 521.239,A 0.000,B 0.000,C 90.000,E1 223.095} C_DIS
LIN {X 0.007,Y -147.216,Z 521.214,A 0.000,B 0.000,C 90.000,E1 218.543} C_DIS
LIN {X -0.024,Y -145.238,Z 521.194,A 0.000,B 0.000,C 90.000,E1 214.898} C_DIS
LIN {X 0.017,Y -142.360,Z 521.163,A 0.000,B 0.000,C 90.000,E1 209.361} C_DIS
LIN {X 0.014,Y -141.746,Z 521.153,A 0.000,B 0.000,C 90.000,E1 207.513} C_DIS
LIN {X -0.059,Y -139.491,Z 521.117,A 0.000,B 0.000,C 90.000,E1 201.046} C_DIS
LIN {X -0.022,Y -138.995,Z 521.101,A 0.000,B 0.000,C 90.000,E1 198.236} C_DIS
LIN {X -0.066,Y -138.336,Z 521.055,A 0.000,B 0.000,C 90.000,E1 189.849} C_DIS
LIN {X -0.044,Y -139.415,Z 521.008,A 0.000,B 0.000,C 90.000,E1 181.432} C_DIS
LIN {X 0.009,Y -141.331,Z 520.972,A 0.000,B 0.000,C 90.000,E1 174.894} C_DIS
LIN {X -0.033,Y -142.688,Z 520.956,A 0.000,B 0.000,C 90.000,E1 172.129} C_DIS
LIN {X -0.055,Y -145.050,Z 520.931,A 0.000,B 0.000,C 90.000,E1 167.521} C_DIS
LIN {X 0.084,Y -147.675,Z 520.910,A 0.000,B 0.000,C 90.000,E1 163.795} C_DIS
LIN {X -0.023,Y -150.318,Z 520.890,A 0.000,B 0.000,C 90.000,E1 160.188} C_DIS
LIN {X 0.049,Y -153.732,Z 520.870,A 0.000,B 0.000,C 90.000,E1 156.538} C_DIS
LIN {X 0.040,Y -157.146,Z 520.850,A 0.000,B 0.000,C 90.000,E1 152.948} C_DIS
LIN {X -0.025,Y -161.295,Z 520.830,A 0.000,B 0.000,C 90.000,E1 149.410} C_DIS
LIN {X -0.008,Y -164.412,Z 520.815,A 0.000,B 0.000,C 90.000,E1 146.755} C_DIS
LIN {X -0.011,Y -169.093,Z 520.796,A 0.000,B 0.000,C 90.000,E1 143.256} C_DIS
LIN {X -0.060,Y -171.650,Z 520.786,A 0.000,B 0.000,C 90.000,E1 141.537} C_DIS
LIN {X -0.014,Y -176.613,Z 520.767,A 0.000,B 0.000,C 90.000,E1 138.081} C_DIS
LIN {X -0.013,Y -180.911,Z 520.753,A 0.000,B 0.000,C 90.000,E1 135.526} C_DIS
LIN {X -0.022,Y -186.327,Z 520.734,A 0.000,B 0.000,C 90.000,E1 132.162} C_DIS
LIN {X 0.030,Y -191.433,Z 520.719,A 0.000,B 0.000,C 90.000,E1 129.358} C_DIS
LIN {X 0.075,Y -192.283,Z 520.716,A 0.000,B 0.000,C 90.000,E1 128.830} C_DIS
LIN {X 0.059,Y -288.959,Z 520.716,A 0.000,B 0.000,C 90.000,E1 128.830} C_DIS
LIN {X -0.050,Y -293.122,Z 520.715,A 0.000,B 0.000,C 90.000,E1 128.749} C_DIS
LIN {X 0.025,Y -296.220,Z 520.714,A 0.000,B 0.000,C 90.000,E1 128.543} C_DIS
LIN {X -0.023,Y -299.879,Z 520.712,A 0.000,B 0.000,C 90.000,E1 128.177} C_DIS
LIN {X -0.062,Y -303.396,Z 520.709,A 0.000,B 0.000,C 90.000,E1 127.604} C_DIS
LIN {X 0.129,Y -304.803,Z 520.707,A 0.000,B 0.000,C 90.000,E1 127.237} C_DIS
LIN {X -0.108,Y -305.911,Z 520.705,A 0.000,B 0.000,C 90.000,E1 126.950} C_DIS
LIN {X 0.061,Y -315.758,Z 520.687,A 0.000,B 0.000,C 90.000,E1 123.658} C_DIS
LIN {X -0.049,Y -325.919,Z 520.671,A 0.000,B 0.000,C 90.000,E1 120.797} C_DIS
LIN {X -0.098,Y -337.421,Z 520.655,A 0.000,B 0.000,C 90.000,E1 117.975} C_DIS
LIN {X -0.133,Y -350.365,Z 520.640,A 0.000,B 0.000,C 90.000,E1 115.207} C_DIS
LIN {X 0.012,Y -363.177,Z 520.627,A 0.000,B 0.000,C 90.000,E1 112.770} C_DIS
LIN {X -0.130,Y -377.314,Z 520.613,A 0.000,B 0.000,C 90.000,E1 110.429} C_DIS
LIN {X -0.061,Y -392.880,Z 520.601,A 0.000,B 0.000,C 90.000,E1 108.109} C_DIS
LIN {X 0.033,Y -409.987,Z 520.588,A 0.000,B 0.000,C 90.000,E1 105.843} C_DIS
LIN {X 0.053,Y -428.763,Z 520.576,A 0.000,B 0.000,C 90.000,E1 103.647} C_DIS
LIN {X -0.108,Y -448.785,Z 520.564,A 0.000,B 0.000,C 90.000,E1 101.591} C_DIS
LIN {X 0.022,Y -469.377,Z 520.554,A 0.000,B 0.000,C 90.000,E1 99.670} C_DIS
LIN {X 0.210,Y -477.242,Z 520.550,A 0.000,B 0.000,C 90.000,E1 98.973} C_DIS
LIN {X -0.221,Y -479.487,Z 520.549,A 0.000,B 0.000,C 90.000,E1 98.803} C_DIS
LIN {X -0.106,Y -481.192,Z 520.548,A 0.000,B 0.000,C 90.000,E1 98.568} C_DIS
LIN {X 0.246,Y -482.663,Z 520.546,A 0.000,B 0.000,C 90.000,E1 98.276} C_DIS
LIN {X 0.052,Y -483.761,Z 520.545,A 0.000,B 0.000,C 90.000,E1 98.049} C_DIS
LIN {X -0.250,Y -485.060,Z 520.542,A 0.000,B 0.000,C 90.000,E1 97.587} C_DIS
LIN {X -0.064,Y -485.335,Z 520.539,A 0.000,B 0.000,C 90.000,E1 97.068} C_DIS
LIN {X 0.131,Y -484.632,Z 520.536,A 0.000,B 0.000,C 90.000,E1 96.549} C_DIS
LIN {X -0.154,Y -482.832,Z 520.534,A 0.000,B 0.000,C 90.000,E1 96.087} C_DIS
LIN {X 0.206,Y -481.413,Z 520.532,A 0.000,B 0.000,C 90.000,E1 95.796} C_DIS
LIN {X 0.022,Y -473.489,Z 520.527,A 0.000,B 0.000,C 90.000,E1 94.821} C_DIS
LIN {X 0.126,Y -459.840,Z 520.517,A 0.000,B 0.000,C 90.000,E1 93.037} C_DIS
LIN {X -0.069,Y -450.997,Z 520.510,A 0.000,B 0.000,C 90.000,E1 91.776} C_DIS
LIN {X 0.161,Y -438.245,Z 520.498,A 0.000,B 0.000,C 90.000,E1 89.656} C_DIS
LIN {X -0.030,Y -426.908,Z 520.488,A 0.000,B 0.000,C 90.000,E1 87.822} C_DIS
LIN {X 0.178,Y -412.515,Z 520.474,A 0.000,B 0.000,C 90.000,E1 85.355} C_DIS
LIN {X 0.022,Y -399.972,Z 520.462,A 0.000,B 0.000,C 90.000,E1 83.166} C_DIS
LIN {X 0.023,Y -389.030,Z 520.451,A 0.000,B 0.000,C 90.000,E1 81.197} C_DIS
LIN {X -0.137,Y -378.087,Z 520.440,A 0.000,B 0.000,C 90.000,E1 79.218} C_DIS
LIN {X -0.095,Y -365.686,Z 520.427,A 0.000,B 0.000,C 90.000,E1 76.881} C_DIS
LIN {X -0.144,Y -353.163,Z 520.412,A 0.000,B 0.000,C 90.000,E1 74.212} C_DIS
LIN {X -0.005,Y -343.430,Z 520.399,A 0.000,B 0.000,C 90.000,E1 71.764} C_DIS
LIN {X 0.083,Y -332.647,Z 520.382,A 0.000,B 0.000,C 90.000,E1 68.666} C_DIS
LIN {X 0.046,Y -322.633,Z 520.364,A 0.000,B 0.000,C 90.000,E1 65.537} C_DIS
LIN {X -0.008,Y -314.942,Z 520.350,A 0.000,B 0.000,C 90.000,E1 62.999} C_DIS
LIN {X 0.025,Y -307.273,Z 520.336,A 0.000,B 0.000,C 90.000,E1 60.411} C_DIS
LIN {X 0.098,Y -297.769,Z 520.317,A 0.000,B 0.000,C 90.000,E1 57.120} C_DIS
LIN {X 0.114,Y -288.781,Z 520.299,A 0.000,B 0.000,C 90.000,E1 53.783} C_DIS
LIN {X 0.006,Y -283.552,Z 520.288,A 0.000,B 0.000,C 90.000,E1 51.778} C_DIS
LIN {X -0.064,Y -278.040,Z 520.276,A 0.000,B 0.000,C 90.000,E1 49.747} C_DIS
LIN {X -0.041,Y -274.083,Z 520.269,A 0.000,B 0.000,C 90.000,E1 48.366} C_DIS
LIN {X 0.015,Y -268.674,Z 520.259,A 0.000,B 0.000,C 90.000,E1 46.620} C_DIS
LIN {X 0.144,Y -262.923,Z 520.249,A 0.000,B 0.000,C 90.000,E1 44.838} C_DIS
LIN {X 0.053,Y -254.735,Z 520.235,A 0.000,B 0.000,C 90.000,E1 42.366} C_DIS
LIN {X 0.006,Y -244.518,Z 520.217,A 0.000,B 0.000,C 90.000,E1 39.116} C_DIS
LIN {X -0.011,Y -236.152,Z 520.201,A 0.000,B 0.000,C 90.000,E1 36.171} C_DIS
LIN {X 0.019,Y -228.562,Z 520.184,A 0.000,B 0.000,C 90.000,E1 33.166} C_DIS
LIN {X -0.010,Y -221.727,Z 520.167,A 0.000,B 0.000,C 90.000,E1 30.129} C_DIS
LIN {X -0.049,Y -215.735,Z 520.150,A 0.000,B 0.000,C 90.000,E1 27.052} C_DIS
LIN {X 0.051,Y -210.560,Z 520.133,A 0.000,B 0.000,C 90.000,E1 23.898} C_DIS
LIN {X 0.065,Y -205.292,Z 520.111,A 0.000,B 0.000,C 90.000,E1 19.939} C_DIS
LIN {X -0.037,Y -201.101,Z 520.089,A 0.000,B 0.000,C 90.000,E1 15.969} C_DIS
LIN {X -0.053,Y -197.367,Z 520.062,A 0.000,B 0.000,C 90.000,E1 11.130} C_DIS
LIN {X 0.050,Y -194.697,Z 520.026,A 0.000,B 0.000,C 90.000,E1 4.588} C_DIS
LIN {X 0.004,Y -196.288,Z 519.961,A 0.000,B 0.000,C 90.000,E1 352.996} C_DIS
LIN {X 0.008,Y -199.368,Z 519.934,A 0.000,B 0.000,C 90.000,E1 348.117} C_DIS
LIN {X -0.068,Y -202.985,Z 519.912,A 0.000,B 0.000,C 90.000,E1 344.102} C_DIS
LIN {X 0.065,Y -207.426,Z 519.889,A 0.000,B 0.000,C 90.000,E1 340.061} C_DIS
LIN {X 0.051,Y -212.640,Z 519.867,A 0.000,B 0.000,C 90.000,E1 336.102} C_DIS
LIN {X -0.131,Y -218.497,Z 519.846,A 0.000,B 0.000,C 90.000,E1 332.231} C_DIS
LIN {X -0.005,Y -224.865,Z 519.824,A 0.000,B 0.000,C 90.000,E1 328.329} C_DIS
LIN {X 0.033,Y -230.524,Z 519.807,A 0.000,B 0.000,C 90.000,E1 325.261} C_DIS
LIN {X 0.022,Y -237.935,Z 519.786,A 0.000,B 0.000,C 90.000,E1 321.492} C_DIS
LIN {X -0.051,Y -246.266,Z 519.765,A 0.000,B 0.000,C 90.000,E1 317.796} C_DIS
LIN {X 0.108,Y -255.689,Z 519.745,A 0.000,B 0.000,C 90.000,E1 314.109} C_DIS
LIN {X 0.089,Y -266.349,Z 519.725,A 0.000,B 0.000,C 90.000,E1 310.539} C_DIS
LIN {X -0.081,Y -278.319,Z 519.706,A 0.000,B 0.000,C 90.000,E1 307.076} C_DIS
LIN {X 0.074,Y -291.580,Z 519.687,A 0.000,B 0.000,C 90.000,E1 303.627} C_DIS
LIN {X -0.170,Y -304.442,Z 519.670,A 0.000,B 0.000,C 90.000,E1 300.669} C_DIS
LIN {X -0.023,Y -319.921,Z 519.652,A 0.000,B 0.000,C 90.000,E1 297.385} C_DIS
LIN {X 0.040,Y -330.105,Z 519.641,A 0.000,B 0.000,C 90.000,E1 295.463} C_DIS
LIN {X 0.158,Y -347.304,Z 519.626,A 0.000,B 0.000,C 90.000,E1 292.642} C_DIS
LIN {X -0.010,Y -364.350,Z 519.612,A 0.000,B 0.000,C 90.000,E1 290.248} C_DIS
LIN {X 0.122,Y -383.028,Z 519.599,A 0.000,B 0.000,C 90.000,E1 287.873} C_DIS
LIN {X -0.062,Y -400.001,Z 519.588,A 0.000,B 0.000,C 90.000,E1 285.898} C_DIS
LIN {X 0.023,Y -417.317,Z 519.578,A 0.000,B 0.000,C 90.000,E1 283.953} C_DIS
LIN {X 0.190,Y -429.482,Z 519.570,A 0.000,B 0.000,C 90.000,E1 282.591} C_DIS
LIN {X -0.122,Y -441.200,Z 519.563,A 0.000,B 0.000,C 90.000,E1 281.299} C_DIS
LIN {X -0.200,Y -450.170,Z 519.557,A 0.000,B 0.000,C 90.000,E1 280.254} C_DIS
LIN {X -0.169,Y -458.369,Z 519.551,A 0.000,B 0.000,C 90.000,E1 279.208} C_DIS
LIN {X 0.135,Y -463.919,Z 519.547,A 0.000,B 0.000,C 90.000,E1 278.398} C_DIS
LIN {X 0.026,Y -468.943,Z 519.542,A 0.000,B 0.000,C 90.000,E1 277.644} C_DIS
LIN {X -0.039,Y -473.479,Z 519.538,A 0.000,B 0.000,C 90.000,E1 276.891} C_DIS
LIN {X 0.207,Y -478.729,Z 519.533,A 0.000,B 0.000,C 90.000,E1 275.853} C_DIS
LIN {X 0.171,Y -482.007,Z 519.529,A 0.000,B 0.000,C 90.000,E1 275.106} C_DIS
LIN {X -0.144,Y -483.747,Z 519.526,A 0.000,B 0.000,C 90.000,E1 274.645} C_DIS
LIN {X -0.007,Y -485.210,Z 519.523,A 0.000,B 0.000,C 90.000,E1 274.131} C_DIS
LIN {X 0.175,Y -486.325,Z 519.520,A 0.000,B 0.000,C 90.000,E1 273.612} C_DIS
LIN {X -0.123,Y -487.113,Z 519.517,A 0.000,B 0.000,C 90.000,E1 273.151} C_DIS
LIN {X 0.045,Y -487.531,Z 519.515,A 0.000,B 0.000,C 90.000,E1 272.636} C_DIS
LIN {X 0.221,Y -487.644,Z 519.512,A 0.000,B 0.000,C 90.000,E1 272.121} C_DIS
LIN {X -0.072,Y -487.376,Z 519.509,A 0.000,B 0.000,C 90.000,E1 271.661} C_DIS
LIN {X 0.107,Y -486.718,Z 519.506,A 0.000,B 0.000,C 90.000,E1 271.146} C_DIS
LIN {X -0.201,Y -485.619,Z 519.504,A 0.000,B 0.000,C 90.000,E1 270.688} C_DIS
LIN {X -0.025,Y -483.946,Z 519.501,A 0.000,B 0.000,C 90.000,E1 270.172} C_DIS
LIN {X -0.182,Y -482.929,Z 519.500,A 0.000,B 0.000,C 90.000,E1 269.943} C_DIS
LIN {X -0.021,Y -480.309,Z 519.497,A 0.000,B 0.000,C 90.000,E1 269.427} C_DIS
LIN {X 0.122,Y -476.908,Z 519.494,A 0.000,B 0.000,C 90.000,E1 268.912} C_DIS
LIN {X -0.049,Y -474.900,Z 519.493,A 0.000,B 0.000,C 90.000,E1 268.682} C_DIS
LIN {X 0.079,Y -469.930,Z 519.490,A 0.000,B 0.000,C 90.000,E1 268.165} C_DIS
LIN {X -0.017,Y -467.123,Z 519.489,A 0.000,B 0.000,C 90.000,E1 267.936} C_DIS
LIN {X -0.113,Y -463.970,Z 519.487,A 0.000,B 0.000,C 90.000,E1 267.707} C_DIS
LIN {X -0.228,Y -457.403,Z 519.485,A 0.000,B 0.000,C 90.000,E1 267.306} C_DIS
LIN {X 0.202,Y -450.238,Z 519.483,A 0.000,B 0.000,C 90.000,E1 266.906} C_DIS
LIN {X -0.107,Y -443.549,Z 519.481,A 0.000,B 0.000,C 90.000,E1 266.674} C_DIS
LIN {X -0.198,Y -436.177,Z 519.480,A 0.000,B 0.000,C 90.000,E1 266.445} C_DIS
LIN {X 0.077,Y -428.626,Z 519.479,A 0.000,B 0.000,C 90.000,E1 266.216} C_DIS
LIN {X -0.157,Y -419.632,Z 519.478,A 0.000,B 0.000,C 90.000,E1 266.102} C_DIS
LIN {X 0.160,Y -411.594,Z 519.478,A 0.000,B 0.000,C 90.000,E1 265.988} C_DIS
LIN {X 0.023,Y -405.687,Z 519.478,A 0.000,B 0.000,C 90.000,E1 265.988} C_DIS
LIN {X -0.009,Y -180.919,Z 519.478,A 0.000,B 0.000,C 90.000,E1 265.988} C_DIS
LIN {X 0.047,Y -180.854,Z 519.472,A 0.000,B 0.000,C 90.000,E1 264.951} C_DIS
LIN {X -0.053,Y -178.904,Z 519.443,A 0.000,B 0.000,C 90.000,E1 259.746} C_DIS
LIN {X 0.027,Y -175.947,Z 519.415,A 0.000,B 0.000,C 90.000,E1 254.629} C_DIS
LIN {X -0.026,Y -175.409,Z 519.410,A 0.000,B 0.000,C 90.000,E1 253.795} C_DIS
LIN {X -0.023,Y -172.174,Z 519.386,A 0.000,B 0.000,C 90.000,E1 249.518} C_DIS
LIN {X 0.017,Y -171.644,Z 519.381,A 0.000,B 0.000,C 90.000,E1 248.646} C_DIS
LIN {X 0.011,Y -167.867,Z 519.357,A 0.000,B 0.000,C 90.000,E1 244.332} C_DIS
LIN {X -0.046,Y -166.601,Z 519.348,A 0.000,B 0.000,C 90.000,E1 242.615} C_DIS
LIN {X -0.051,Y -162.590,Z 519.323,A 0.000,B 0.000,C 90.000,E1 238.250} C_DIS
LIN {X -0.077,Y -161.274,Z 519.314,A 0.000,B 0.000,C 90.000,E1 236.501} C_DIS
LIN {X -0.042,Y -157.274,Z 519.289,A 0.000,B 0.000,C 90.000,E1 232.065} C_DIS
LIN {X -0.019,Y -155.993,Z 519.279,A 0.000,B 0.000,C 90.000,E1 230.275} C_DIS
LIN {X -0.057,Y -152.250,Z 519.254,A 0.000,B 0.000,C 90.000,E1 225.810} C_DIS
LIN {X -0.035,Y -150.490,Z 519.239,A 0.000,B 0.000,C 90.000,E1 223.095} C_DIS
LIN {X -0.006,Y -147.214,Z 519.214,A 0.000,B 0.000,C 90.000,E1 218.543} C_DIS
LIN {X -0.035,Y -145.235,Z 519.194,A 0.000,B 0.000,C 90.000,E1 214.898} C_DIS
LIN {X 0.075,Y -142.358,Z 519.163,A 0.000,B 0.000,C 90.000,E1 209.333} C_DIS
LIN {X 0.003,Y -141.745,Z 519.153,A 0.000,B 0.000,C 90.000,E1 207.513} C_DIS
LIN {X -0.071,Y -139.491,Z 519.117,A 0.000,B 0.000,C 90.000,E1 201.046} C_DIS
LIN {X -0.033,Y -138.993,Z 519.101,A 0.000,B 0.000,C 90.000,E1 198.236} C_DIS
LIN {X 0.060,Y -138.336,Z 519.055,A 0.000,B 0.000,C 90.000,E1 189.792} C_DIS
LIN {X -0.055,Y -139.416,Z 519.008,A 0.000,B 0.000,C 90.000,E1 181.432} C_DIS
LIN {X -0.002,Y -141.333,Z 518.972,A 0.000,B 0.000,C 90.000,E1 174.894} C_DIS
LIN {X -0.045,Y -142.689,Z 518.956,A 0.000,B 0.000,C 90.000,E1 172.129} C_DIS
LIN {X 0.075,Y -145.052,Z 518.931,A 0.000,B 0.000,C 90.000,E1 167.465} C_DIS
LIN {X 0.072,Y -147.677,Z 518.910,A 0.000,B 0.000,C 90.000,E1 163.795} C_DIS
LIN {X -0.035,Y -150.322,Z 518.890,A 0.000,B 0.000,C 90.000,E1 160.188} C_DIS
LIN {X 0.037,Y -153.738,Z 518.870,A 0.000,B 0.000,C 90.000,E1 156.538} C_DIS
LIN {X 0.028,Y -157.151,Z 518.850,A 0.000,B 0.000,C 90.000,E1 152.948} C_DIS
LIN {X -0.038,Y -161.301,Z 518.830,A 0.000,B 0.000,C 90.000,E1 149.410} C_DIS
LIN {X -0.020,Y -164.416,Z 518.815,A 0.000,B 0.000,C 90.000,E1 146.755} C_DIS
LIN {X -0.024,Y -169.099,Z 518.796,A 0.000,B 0.000,C 90.000,E1 143.256} C_DIS
LIN {X -0.073,Y -171.655,Z 518.786,A 0.000,B 0.000,C 90.000,E1 141.537} C_DIS
LIN {X -0.027,Y -176.619,Z 518.767,A 0.000,B 0.000,C 90.000,E1 138.081} C_DIS
LIN {X 0.100,Y -180.917,Z 518.753,A 0.000,B 0.000,C 90.000,E1 135.486} C_DIS
LIN {X -0.035,Y -186.335,Z 518.734,A 0.000,B 0.000,C 90.000,E1 132.162} C_DIS
LIN {X 0.031,Y -190.968,Z 518.720,A 0.000,B 0.000,C 90.000,E1 129.644} C_DIS
LIN {X -0.011,Y -192.326,Z 518.716,A 0.000,B 0.000,C 90.000,E1 128.830} C_DIS
LIN {X -0.052,Y -289.347,Z 518.716,A 0.000,B 0.000,C 90.000,E1 128.830} C_DIS
LIN {X 0.033,Y -292.271,Z 518.715,A 0.000,B 0.000,C 90.000,E1 128.749} C_DIS
LIN {X -0.017,Y -297.925,Z 518.713,A 0.000,B 0.000,C 90.000,E1 128.382} C_DIS
LIN {X -0.068,Y -300.988,Z 518.711,A 0.000,B 0.000,C 90.000,E1 128.016} C_DIS
LIN {X 0.122,Y -302.934,Z 518.709,A 0.000,B 0.000,C 90.000,E1 127.649} C_DIS
LIN {X -0.114,Y -304.447,Z 518.707,A 0.000,B 0.000,C 90.000,E1 127.363} C_DIS
LIN {X 0.086,Y -305.633,Z 518.706,A 0.000,B 0.000,C 90.000,E1 126.996} C_DIS
LIN {X 0.035,Y -316.538,Z 518.686,A 0.000,B 0.000,C 90.000,E1 123.420} C_DIS
LIN {X 0.046,Y -326.807,Z 518.670,A 0.000,B 0.000,C 90.000,E1 120.541} C_DIS
LIN {X 0.031,Y -338.426,Z 518.654,A 0.000,B 0.000,C 90.000,E1 117.719} C_DIS
LIN {X 0.029,Y -351.495,Z 518.639,A 0.000,B 0.000,C 90.000,E1 114.951} C_DIS
LIN {X 0.208,Y -364.427,Z 518.625,A 0.000,B 0.000,C 90.000,E1 112.514} C_DIS
LIN {X 0.098,Y -378.695,Z 518.612,A 0.000,B 0.000,C 90.000,E1 110.174} C_DIS
LIN {X 0.081,Y -394.400,Z 518.599,A 0.000,B 0.000,C 90.000,E1 107.873} C_DIS
LIN {X -0.172,Y -411.659,Z 518.587,A 0.000,B 0.000,C 90.000,E1 105.662} C_DIS
LIN {X -0.119,Y -430.593,Z 518.575,A 0.000,B 0.000,C 90.000,E1 103.467} C_DIS
LIN {X 0.185,Y -450.681,Z 518.563,A 0.000,B 0.000,C 90.000,E1 101.366} C_DIS
LIN {X 0.001,Y -471.322,Z 518.553,A 0.000,B 0.000,C 90.000,E1 99.500} C_DIS
LIN {X -0.236,Y -479.004,Z 518.549,A 0.000,B 0.000,C 90.000,E1 98.859} C_DIS
LIN {X -0.203,Y -480.933,Z 518.548,A 0.000,B 0.000,C 90.000,E1 98.624} C_DIS
LIN {X -0.242,Y -482.410,Z 518.547,A 0.000,B 0.000,C 90.000,E1 98.398} C_DIS
LIN {X 0.115,Y -483.618,Z 518.545,A 0.000,B 0.000,C 90.000,E1 98.106} C_DIS
LIN {X -0.007,Y -484.500,Z 518.544,A 0.000,B 0.000,C 90.000,E1 97.871} C_DIS
LIN {X 0.174,Y -485.437,Z 518.541,A 0.000,B 0.000,C 90.000,E1 97.352} C_DIS
LIN {X -0.118,Y -485.384,Z 518.538,A 0.000,B 0.000,C 90.000,E1 96.891} C_DIS
LIN {X 0.076,Y -484.331,Z 518.535,A 0.000,B 0.000,C 90.000,E1 96.372} C_DIS
LIN {X -0.094,Y -483.382,Z 518.534,A 0.000,B 0.000,C 90.000,E1 96.144} C_DIS
LIN {X -0.211,Y -482.092,Z 518.533,A 0.000,B 0.000,C 90.000,E1 95.910} C_DIS
LIN {X 0.095,Y -480.365,Z 518.531,A 0.000,B 0.000,C 90.000,E1 95.625} C_DIS
LIN {X 0.203,Y -460.588,Z 518.517,A 0.000,B 0.000,C 90.000,E1 93.094} C_DIS
LIN {X 0.006,Y -451.673,Z 518.510,A 0.000,B 0.000,C 90.000,E1 91.835} C_DIS
LIN {X -0.004,Y -437.218,Z 518.497,A 0.000,B 0.000,C 90.000,E1 89.484} C_DIS
LIN {X 0.213,Y -425.854,Z 518.487,A 0.000,B 0.000,C 90.000,E1 87.593} C_DIS
LIN {X 0.005,Y -411.496,Z 518.473,A 0.000,B 0.000,C 90.000,E1 85.179} C_DIS
LIN {X -0.124,Y -397.390,Z 518.459,A 0.000,B 0.000,C 90.000,E1 82.704} C_DIS
LIN {X -0.178,Y -386.432,Z 518.448,A 0.000,B 0.000,C 90.000,E1 80.735} C_DIS
LIN {X -0.037,Y -377.022,Z 518.439,A 0.000,B 0.000,C 90.000,E1 78.993} C_DIS
LIN {X 0.048,Y -364.712,Z 518.426,A 0.000,B 0.000,C 90.000,E1 76.645} C_DIS
LIN {X -0.071,Y -353.572,Z 518.413,A 0.000,B 0.000,C 90.000,E1 74.283} C_DIS
LIN {X 0.174,Y -343.782,Z 518.399,A 0.000,B 0.000,C 90.000,E1 71.819} C_DIS
LIN {X -0.053,Y -331.916,Z 518.380,A 0.000,B 0.000,C 90.000,E1 68.465} C_DIS
LIN {X 0.063,Y -321.960,Z 518.363,A 0.000,B 0.000,C 90.000,E1 65.305} C_DIS
LIN {X 0.125,Y -314.222,Z 518.349,A 0.000,B 0.000,C 90.000,E1 62.743} C_DIS
LIN {X -0.080,Y -308.465,Z 518.338,A 0.000,B 0.000,C 90.000,E1 60.845} C_DIS
LIN {X 0.092,Y -300.789,Z 518.323,A 0.000,B 0.000,C 90.000,E1 58.201} C_DIS
LIN {X 0.042,Y -291.576,Z 518.305,A 0.000,B 0.000,C 90.000,E1 54.895} C_DIS
LIN {X 0.105,Y -284.576,Z 518.290,A 0.000,B 0.000,C 90.000,E1 52.190} C_DIS
LIN {X 0.092,Y -279.140,Z 518.279,A 0.000,B 0.000,C 90.000,E1 50.150} C_DIS
LIN {X 0.122,Y -275.285,Z 518.271,A 0.000,B 0.000,C 90.000,E1 48.771} C_DIS
LIN {X 0.108,Y -271.086,Z 518.263,A 0.000,B 0.000,C 90.000,E1 47.391} C_DIS
LIN {X 0.096,Y -265.497,Z 518.254,A 0.000,B 0.000,C 90.000,E1 45.648} C_DIS
LIN {X 0.068,Y -257.299,Z 518.240,A 0.000,B 0.000,C 90.000,E1 43.176} C_DIS
LIN {X 0.066,Y -246.977,Z 518.222,A 0.000,B 0.000,C 90.000,E1 39.930} C_DIS
LIN {X -0.106,Y -237.374,Z 518.204,A 0.000,B 0.000,C 90.000,E1 36.664} C_DIS
LIN {X -0.042,Y -229.658,Z 518.187,A 0.000,B 0.000,C 90.000,E1 33.658} C_DIS
LIN {X 0.077,Y -222.706,Z 518.170,A 0.000,B 0.000,C 90.000,E1 30.590} C_DIS
LIN {X 0.060,Y -216.571,Z 518.153,A 0.000,B 0.000,C 90.000,E1 27.513} C_DIS
LIN {X 0.078,Y -211.276,Z 518.136,A 0.000,B 0.000,C 90.000,E1 24.387} C_DIS
LIN {X -0.083,Y -205.852,Z 518.114,A 0.000,B 0.000,C 90.000,E1 20.482} C_DIS
LIN {X 0.083,Y -201.543,Z 518.091,A 0.000,B 0.000,C 90.000,E1 16.441} C_DIS
LIN {X -0.114,Y -197.663,Z 518.065,A 0.000,B 0.000,C 90.000,E1 11.658} C_DIS
LIN {X 0.075,Y -194.957,Z 518.033,A 0.000,B 0.000,C 90.000,E1 5.910} C_DIS
LIN {X 0.001,Y -196.186,Z 517.961,A 0.000,B 0.000,C 90.000,E1 352.996} C_DIS
LIN {X 0.036,Y -199.874,Z 517.930,A 0.000,B 0.000,C 90.000,E1 347.297} C_DIS
LIN {X 0.027,Y -203.699,Z 517.907,A 0.000,B 0.000,C 90.000,E1 343.268} C_DIS
LIN {X 0.055,Y -208.284,Z 517.885,A 0.000,B 0.000,C 90.000,E1 339.263} C_DIS
LIN {X 0.063,Y -213.639,Z 517.863,A 0.000,B 0.000,C 90.000,E1 335.305} C_DIS
LIN {X 0.102,Y -219.607,Z 517.841,A 0.000,B 0.000,C 90.000,E1 331.385} C_DIS
LIN {X 0.074,Y -226.131,Z 517.820,A 0.000,B 0.000,C 90.000,E1 327.533} C_DIS
LIN {X 0.081,Y -231.856,Z 517.803,A 0.000,B 0.000,C 90.000,E1 324.482} C_DIS
LIN {X 0.076,Y -239.447,Z 517.782,A 0.000,B 0.000,C 90.000,E1 320.723} C_DIS
LIN {X 0.058,Y -247.980,Z 517.761,A 0.000,B 0.000,C 90.000,E1 317.025} C_DIS
LIN {X -0.099,Y -256.663,Z 517.743,A 0.000,B 0.000,C 90.000,E1 313.785} C_DIS
LIN {X 0.106,Y -267.451,Z 517.723,A 0.000,B 0.000,C 90.000,E1 310.172} C_DIS
LIN {X -0.029,Y -279.574,Z 517.704,A 0.000,B 0.000,C 90.000,E1 306.710} C_DIS
LIN {X 0.003,Y -292.986,Z 517.685,A 0.000,B 0.000,C 90.000,E1 303.293} C_DIS
LIN {X 0.060,Y -305.915,Z 517.668,A 0.000,B 0.000,C 90.000,E1 300.285} C_DIS
LIN {X -0.013,Y -321.556,Z 517.650,A 0.000,B 0.000,C 90.000,E1 297.052} C_DIS
LIN {X -0.066,Y -331.945,Z 517.640,A 0.000,B 0.000,C 90.000,E1 295.155} C_DIS
LIN {X 0.111,Y -349.358,Z 517.624,A 0.000,B 0.000,C 90.000,E1 292.333} C_DIS
LIN {X -0.006,Y -366.597,Z 517.611,A 0.000,B 0.000,C 90.000,E1 289.939} C_DIS
LIN {X 0.192,Y -387.904,Z 517.596,A 0.000,B 0.000,C 90.000,E1 287.275} C_DIS
LIN {X -0.104,Y -410.020,Z 517.582,A 0.000,B 0.000,C 90.000,E1 284.773} C_DIS
LIN {X 0.182,Y -422.540,Z 517.574,A 0.000,B 0.000,C 90.000,E1 283.355} C_DIS
LIN {X 0.073,Y -432.218,Z 517.568,A 0.000,B 0.000,C 90.000,E1 282.299} C_DIS
LIN {X 0.195,Y -443.921,Z 517.561,A 0.000,B 0.000,C 90.000,E1 280.950} C_DIS
LIN {X 0.158,Y -452.701,Z 517.555,A 0.000,B 0.000,C 90.000,E1 279.905} C_DIS
LIN {X -0.048,Y -458.781,Z 517.551,A 0.000,B 0.000,C 90.000,E1 279.151} C_DIS
LIN {X -0.197,Y -464.302,Z 517.547,A 0.000,B 0.000,C 90.000,E1 278.398} C_DIS
LIN {X 0.000,Y -470.897,Z 517.541,A 0.000,B 0.000,C 90.000,E1 277.352} C_DIS
LIN {X -0.111,Y -475.203,Z 517.537,A 0.000,B 0.000,C 90.000,E1 276.606} C_DIS
LIN {X -0.125,Y -479.019,Z 517.532,A 0.000,B 0.000,C 90.000,E1 275.853} C_DIS
LIN {X -0.162,Y -482.278,Z 517.528,A 0.000,B 0.000,C 90.000,E1 275.106} C_DIS
LIN {X 0.007,Y -484.025,Z 517.526,A 0.000,B 0.000,C 90.000,E1 274.588} C_DIS
LIN {X 0.146,Y -485.436,Z 517.523,A 0.000,B 0.000,C 90.000,E1 274.073} C_DIS
LIN {X -0.155,Y -486.525,Z 517.520,A 0.000,B 0.000,C 90.000,E1 273.612} C_DIS
LIN {X 0.034,Y -487.287,Z 517.517,A 0.000,B 0.000,C 90.000,E1 273.094} C_DIS
LIN {X 0.203,Y -487.683,Z 517.514,A 0.000,B 0.000,C 90.000,E1 272.579} C_DIS
LIN {X -0.107,Y -487.741,Z 517.512,A 0.000,B 0.000,C 90.000,E1 272.121} C_DIS
LIN {X 0.088,Y -487.458,Z 517.509,A 0.000,B 0.000,C 90.000,E1 271.604} C_DIS
LIN {X -0.219,Y -486.762,Z 517.506,A 0.000,B 0.000,C 90.000,E1 271.146} C_DIS
LIN {X -0.040,Y -485.605,Z 517.503,A 0.000,B 0.000,C 90.000,E1 270.630} C_DIS
LIN {X 0.135,Y -483.891,Z 517.501,A 0.000,B 0.000,C 90.000,E1 270.115} C_DIS
LIN {X -0.022,Y -482.832,Z 517.499,A 0.000,B 0.000,C 90.000,E1 269.885} C_DIS
LIN {X 0.137,Y -480.141,Z 517.497,A 0.000,B 0.000,C 90.000,E1 269.370} C_DIS
LIN {X -0.027,Y -478.526,Z 517.495,A 0.000,B 0.000,C 90.000,E1 269.141} C_DIS
LIN {X 0.107,Y -474.509,Z 517.492,A 0.000,B 0.000,C 90.000,E1 268.625} C_DIS
LIN {X -0.073,Y -472.208,Z 517.491,A 0.000,B 0.000,C 90.000,E1 268.396} C_DIS
LIN {X 0.232,Y -469.542,Z 517.490,A 0.000,B 0.000,C 90.000,E1 268.108} C_DIS
LIN {X 0.083,Y -463.533,Z 517.487,A 0.000,B 0.000,C 90.000,E1 267.650} C_DIS
LIN {X -0.190,Y -460.447,Z 517.486,A 0.000,B 0.000,C 90.000,E1 267.478} C_DIS
LIN {X 0.030,Y -453.627,Z 517.484,A 0.000,B 0.000,C 90.000,E1 267.078} C_DIS
LIN {X -0.092,Y -446.640,Z 517.482,A 0.000,B 0.000,C 90.000,E1 266.788} C_DIS
LIN {X 0.144,Y -439.711,Z 517.481,A 0.000,B 0.000,C 90.000,E1 266.502} C_DIS
LIN {X -0.168,Y -432.342,Z 517.479,A 0.000,B 0.000,C 90.000,E1 266.331} C_DIS
LIN {X -0.134,Y -424.399,Z 517.479,A 0.000,B 0.000,C 90.000,E1 266.159} C_DIS
LIN {X -0.163,Y -413.681,Z 517.478,A 0.000,B 0.000,C 90.000,E1 266.045} C_DIS
LIN {X 0.001,Y -403.434,Z 517.478,A 0.000,B 0.000,C 90.000,E1 265.988} C_DIS
LIN {X -0.035,Y -180.919,Z 517.478,A 0.000,B 0.000,C 90.000,E1 265.988} C_DIS
LIN {X 0.006,Y -180.850,Z 517.472,A 0.000,B 0.000,C 90.000,E1 264.951} C_DIS
LIN {X 0.082,Y -178.898,Z 517.443,A 0.000,B 0.000,C 90.000,E1 259.690} C_DIS
LIN {X -0.013,Y -175.942,Z 517.415,A 0.000,B 0.000,C 90.000,E1 254.629} C_DIS
LIN {X -0.066,Y -175.397,Z 517.410,A 0.000,B 0.000,C 90.000,E1 253.795} C_DIS
LIN {X -0.063,Y -172.165,Z 517.386,A 0.000,B 0.000,C 90.000,E1 249.518} C_DIS
LIN {X -0.024,Y -171.634,Z 517.381,A 0.000,B 0.000,C 90.000,E1 248.646} C_DIS
LIN {X -0.028,Y -167.857,Z 517.357,A 0.000,B 0.000,C 90.000,E1 244.332} C_DIS
LIN {X -0.085,Y -166.589,Z 517.348,A 0.000,B 0.000,C 90.000,E1 242.615} C_DIS
LIN {X 0.049,Y -162.579,Z 517.323,A 0.000,B 0.000,C 90.000,E1 238.201} C_DIS
LIN {X 0.108,Y -161.262,Z 517.314,A 0.000,B 0.000,C 90.000,E1 236.421} C_DIS
LIN {X 0.018,Y -157.263,Z 517.289,A 0.000,B 0.000,C 90.000,E1 232.029} C_DIS
LIN {X -0.056,Y -155.984,Z 517.279,A 0.000,B 0.000,C 90.000,E1 230.275} C_DIS
LIN {X -0.095,Y -152.241,Z 517.254,A 0.000,B 0.000,C 90.000,E1 225.810} C_DIS
LIN {X 0.030,Y -150.481,Z 517.239,A 0.000,B 0.000,C 90.000,E1 223.056} C_DIS
LIN {X -0.041,Y -147.205,Z 517.214,A 0.000,B 0.000,C 90.000,E1 218.543} C_DIS
LIN {X -0.071,Y -145.226,Z 517.194,A 0.000,B 0.000,C 90.000,E1 214.898} C_DIS
LIN {X 0.041,Y -142.352,Z 517.163,A 0.000,B 0.000,C 90.000,E1 209.333} C_DIS
LIN {X -0.033,Y -141.740,Z 517.153,A 0.000,B 0.000,C 90.000,E1 207.513} C_DIS
LIN {X 0.074,Y -139.488,Z 517.117,A 0.000,B 0.000,C 90.000,E1 200.972} C_DIS
LIN {X 0.063,Y -138.989,Z 517.101,A 0.000,B 0.000,C 90.000,E1 198.181} C_DIS
LIN {X 0.024,Y -138.334,Z 517.054,A 0.000,B 0.000,C 90.000,E1 189.792} C_DIS
LIN {X 0.049,Y -139.420,Z 517.008,A 0.000,B 0.000,C 90.000,E1 181.375} C_DIS
LIN {X -0.038,Y -141.339,Z 516.972,A 0.000,B 0.000,C 90.000,E1 174.894} C_DIS
LIN {X 0.060,Y -142.695,Z 516.956,A 0.000,B 0.000,C 90.000,E1 172.072} C_DIS
LIN {X 0.039,Y -145.061,Z 516.930,A 0.000,B 0.000,C 90.000,E1 167.465} C_DIS
LIN {X 0.037,Y -147.687,Z 516.910,A 0.000,B 0.000,C 90.000,E1 163.795} C_DIS
LIN {X -0.071,Y -150.333,Z 516.890,A 0.000,B 0.000,C 90.000,E1 160.188} C_DIS
LIN {X 0.000,Y -153.752,Z 516.870,A 0.000,B 0.000,C 90.000,E1 156.538} C_DIS
LIN {X -0.009,Y -157.165,Z 516.850,A 0.000,B 0.000,C 90.000,E1 152.948} C_DIS
LIN {X -0.076,Y -161.319,Z 516.830,A 0.000,B 0.000,C 90.000,E1 149.410} C_DIS
LIN {X 0.078,Y -164.433,Z 516.815,A 0.000,B 0.000,C 90.000,E1 146.707} C_DIS
LIN {X 0.071,Y -169.119,Z 516.796,A 0.000,B 0.000,C 90.000,E1 143.210} C_DIS
LIN {X 0.021,Y -171.673,Z 516.786,A 0.000,B 0.000,C 90.000,E1 141.492} C_DIS
LIN {X -0.068,Y -176.641,Z 516.767,A 0.000,B 0.000,C 90.000,E1 138.081} C_DIS
LIN {X 0.059,Y -180.938,Z 516.753,A 0.000,B 0.000,C 90.000,E1 135.486} C_DIS
LIN {X 0.047,Y -186.358,Z 516.734,A 0.000,B 0.000,C 90.000,E1 132.123} C_DIS
LIN {X -0.012,Y -190.989,Z 516.720,A 0.000,B 0.000,C 90.000,E1 129.644} C_DIS
LIN {X -0.077,Y -192.359,Z 516.716,A 0.000,B 0.000,C 90.000,E1 128.830} C_DIS
LIN {X -0.151,Y -289.244,Z 516.716,A 0.000,B 0.000,C 90.000,E1 128.830} C_DIS
LIN {X -0.032,Y -292.082,Z 516.715,A 0.000,B 0.000,C 90.000,E1 128.749} C_DIS
LIN {X 0.059,Y -295.668,Z 516.714,A 0.000,B 0.000,C 90.000,E1 128.543} C_DIS
LIN {X -0.084,Y -297.882,Z 516.713,A 0.000,B 0.000,C 90.000,E1 128.382} C_DIS
LIN {X -0.135,Y -300.971,Z 516.711,A 0.000,B 0.000,C 90.000,E1 128.016} C_DIS
LIN {X 0.065,Y -302.920,Z 516.709,A 0.000,B 0.000,C 90.000,E1 127.649} C_DIS
LIN {X 0.081,Y -304.436,Z 516.707,A 0.000,B 0.000,C 90.000,E1 127.317} C_DIS
LIN {X 0.039,Y -305.632,Z 516.706,A 0.000,B 0.000,C 90.000,E1 126.996} C_DIS
LIN {X -0.013,Y -316.546,Z 516.686,A 0.000,B 0.000,C 90.000,E1 123.420} C_DIS
LIN {X -0.003,Y -326.819,Z 516.670,A 0.000,B 0.000,C 90.000,E1 120.541} C_DIS
LIN {X -0.020,Y -338.442,Z 516.654,A 0.000,B 0.000,C 90.000,E1 117.719} C_DIS
LIN {X -0.023,Y -351.515,Z 516.639,A 0.000,B 0.000,C 90.000,E1 114.951} C_DIS
LIN {X 0.153,Y -364.451,Z 516.625,A 0.000,B 0.000,C 90.000,E1 112.514} C_DIS
LIN {X 0.043,Y -378.723,Z 516.612,A 0.000,B 0.000,C 90.000,E1 110.174} C_DIS
LIN {X 0.023,Y -394.434,Z 516.599,A 0.000,B 0.000,C 90.000,E1 107.873} C_DIS
LIN {X 0.165,Y -411.698,Z 516.587,A 0.000,B 0.000,C 90.000,E1 105.607} C_DIS
LIN {X 0.240,Y -430.639,Z 516.575,A 0.000,B 0.000,C 90.000,E1 103.411} C_DIS
LIN {X 0.127,Y -450.729,Z 516.563,A 0.000,B 0.000,C 90.000,E1 101.366} C_DIS
LIN {X -0.055,Y -471.370,Z 516.553,A 0.000,B 0.000,C 90.000,E1 99.500} C_DIS
LIN {X 0.182,Y -479.078,Z 516.549,A 0.000,B 0.000,C 90.000,E1 98.803} C_DIS
LIN {X 0.228,Y -481.021,Z 516.548,A 0.000,B 0.000,C 90.000,E1 98.568} C_DIS
LIN {X 0.204,Y -482.508,Z 516.546,A 0.000,B 0.000,C 90.000,E1 98.341} C_DIS
LIN {X 0.083,Y -483.737,Z 516.545,A 0.000,B 0.000,C 90.000,E1 98.106} C_DIS
LIN {X -0.039,Y -484.634,Z 516.544,A 0.000,B 0.000,C 90.000,E1 97.871} C_DIS
LIN {X 0.144,Y -485.598,Z 516.541,A 0.000,B 0.000,C 90.000,E1 97.352} C_DIS
LIN {X -0.148,Y -485.569,Z 516.538,A 0.000,B 0.000,C 90.000,E1 96.891} C_DIS
LIN {X 0.047,Y -484.544,Z 516.535,A 0.000,B 0.000,C 90.000,E1 96.372} C_DIS
LIN {X -0.122,Y -483.612,Z 516.534,A 0.000,B 0.000,C 90.000,E1 96.144} C_DIS
LIN {X 0.241,Y -482.340,Z 516.533,A 0.000,B 0.000,C 90.000,E1 95.853} C_DIS
LIN {X 0.068,Y -480.638,Z 516.531,A 0.000,B 0.000,C 90.000,E1 95.625} C_DIS
LIN {X 0.184,Y -460.831,Z 516.517,A 0.000,B 0.000,C 90.000,E1 93.094} C_DIS
LIN {X -0.009,Y -451.875,Z 516.510,A 0.000,B 0.000,C 90.000,E1 91.835} C_DIS
LIN {X -0.014,Y -437.371,Z 516.497,A 0.000,B 0.000,C 90.000,E1 89.484} C_DIS
LIN {X 0.207,Y -425.981,Z 516.487,A 0.000,B 0.000,C 90.000,E1 87.593} C_DIS
LIN {X 0.003,Y -411.614,Z 516.473,A 0.000,B 0.000,C 90.000,E1 85.179} C_DIS
LIN {X -0.124,Y -397.523,Z 516.459,A 0.000,B 0.000,C 90.000,E1 82.704} C_DIS
LIN {X -0.174,Y -386.560,Z 516.448,A 0.000,B 0.000,C 90.000,E1 80.735} C_DIS
LIN {X -0.012,Y -375.566,Z 516.437,A 0.000,B 0.000,C 90.000,E1 78.701} C_DIS
LIN {X 0.056,Y -364.802,Z 516.426,A 0.000,B 0.000,C 90.000,E1 76.645} C_DIS
LIN {X -0.062,Y -353.647,Z 516.413,A 0.000,B 0.000,C 90.000,E1 74.283} C_DIS
LIN {X 0.184,Y -343.845,Z 516.399,A 0.000,B 0.000,C 90.000,E1 71.819} C_DIS
LIN {X -0.035,Y -331.964,Z 516.380,A 0.000,B 0.000,C 90.000,E1 68.465} C_DIS
LIN {X 0.083,Y -322.000,Z 516.363,A 0.000,B 0.000,C 90.000,E1 65.305} C_DIS
LIN {X 0.144,Y -314.228,Z 516.349,A 0.000,B 0.000,C 90.000,E1 62.743} C_DIS
LIN {X -0.112,Y -306.518,Z 516.334,A 0.000,B 0.000,C 90.000,E1 60.205} C_DIS
LIN {X -0.094,Y -298.859,Z 516.320,A 0.000,B 0.000,C 90.000,E1 57.582} C_DIS
LIN {X -0.027,Y -289.740,Z 516.301,A 0.000,B 0.000,C 90.000,E1 54.242} C_DIS
LIN {X 0.119,Y -284.495,Z 516.290,A 0.000,B 0.000,C 90.000,E1 52.190} C_DIS
LIN {X -0.110,Y -279.050,Z 516.279,A 0.000,B 0.000,C 90.000,E1 50.194} C_DIS
LIN {X 0.133,Y -275.193,Z 516.271,A 0.000,B 0.000,C 90.000,E1 48.771} C_DIS
LIN {X 0.117,Y -271.007,Z 516.263,A 0.000,B 0.000,C 90.000,E1 47.391} C_DIS
LIN {X 0.104,Y -265.414,Z 516.254,A 0.000,B 0.000,C 90.000,E1 45.648} C_DIS
LIN {X -0.077,Y -256.049,Z 516.238,A 0.000,B 0.000,C 90.000,E1 42.852} C_DIS
LIN {X 0.081,Y -245.812,Z 516.220,A 0.000,B 0.000,C 90.000,E1 39.564} C_DIS
LIN {X -0.103,Y -237.326,Z 516.204,A 0.000,B 0.000,C 90.000,E1 36.664} C_DIS
LIN {X -0.041,Y -229.602,Z 516.187,A 0.000,B 0.000,C 90.000,E1 33.658} C_DIS
LIN {X 0.077,Y -222.645,Z 516.170,A 0.000,B 0.000,C 90.000,E1 30.590} C_DIS
LIN {X 0.059,Y -216.515,Z 516.153,A 0.000,B 0.000,C 90.000,E1 27.513} C_DIS
LIN {X 0.075,Y -211.232,Z 516.136,A 0.000,B 0.000,C 90.000,E1 24.387} C_DIS
LIN {X -0.088,Y -205.821,Z 516.114,A 0.000,B 0.000,C 90.000,E1 20.482} C_DIS
LIN {X 0.079,Y -201.508,Z 516.091,A 0.000,B 0.000,C 90.000,E1 16.441} C_DIS
LIN {X 0.073,Y -197.627,Z 516.065,A 0.000,B 0.000,C 90.000,E1 11.602} C_DIS
LIN {X 0.067,Y -194.907,Z 516.033,A 0.000,B 0.000,C 90.000,E1 5.910} C_DIS
LIN {X -0.004,Y -196.084,Z 515.961,A 0.000,B 0.000,C 90.000,E1 352.996} C_DIS
LIN {X 0.026,Y -199.743,Z 515.929,A 0.000,B 0.000,C 90.000,E1 347.297} C_DIS
LIN {X 0.014,Y -203.565,Z 515.907,A 0.000,B 0.000,C 90.000,E1 343.268} C_DIS
LIN {X 0.037,Y -208.158,Z 515.885,A 0.000,B 0.000,C 90.000,E1 339.263} C_DIS
LIN {X 0.041,Y -213.512,Z 515.863,A 0.000,B 0.000,C 90.000,E1 335.305} C_DIS
LIN {X 0.076,Y -219.485,Z 515.841,A 0.000,B 0.000,C 90.000,E1 331.385} C_DIS
LIN {X 0.042,Y -226.019,Z 515.820,A 0.000,B 0.000,C 90.000,E1 327.533} C_DIS
LIN {X 0.045,Y -231.761,Z 515.803,A 0.000,B 0.000,C 90.000,E1 324.482} C_DIS
LIN {X 0.037,Y -239.367,Z 515.782,A 0.000,B 0.000,C 90.000,E1 320.723} C_DIS
LIN {X 0.015,Y -247.907,Z 515.761,A 0.000,B 0.000,C 90.000,E1 317.025} C_DIS
LIN {X 0.054,Y -257.664,Z 515.741,A 0.000,B 0.000,C 90.000,E1 313.380} C_DIS
LIN {X -0.085,Y -268.578,Z 515.721,A 0.000,B 0.000,C 90.000,E1 309.850} C_DIS
LIN {X -0.144,Y -280.842,Z 515.702,A 0.000,B 0.000,C 90.000,E1 306.377} C_DIS
LIN {X -0.067,Y -294.408,Z 515.683,A 0.000,B 0.000,C 90.000,E1 302.959} C_DIS
LIN {X 0.067,Y -308.913,Z 515.665,A 0.000,B 0.000,C 90.000,E1 299.617} C_DIS
LIN {X -0.066,Y -324.904,Z 515.647,A 0.000,B 0.000,C 90.000,E1 296.411} C_DIS
LIN {X -0.022,Y -333.819,Z 515.638,A 0.000,B 0.000,C 90.000,E1 294.823} C_DIS
LIN {X 0.045,Y -349.381,Z 515.624,A 0.000,B 0.000,C 90.000,E1 292.333} C_DIS
LIN {X -0.005,Y -368.886,Z 515.609,A 0.000,B 0.000,C 90.000,E1 289.631} C_DIS
LIN {X 0.148,Y -390.334,Z 515.594,A 0.000,B 0.000,C 90.000,E1 286.985} C_DIS
LIN {X -0.180,Y -410.073,Z 515.582,A 0.000,B 0.000,C 90.000,E1 284.773} C_DIS
LIN {X 0.120,Y -422.621,Z 515.574,A 0.000,B 0.000,C 90.000,E1 283.355} C_DIS
LIN {X -0.081,Y -432.417,Z 515.568,A 0.000,B 0.000,C 90.000,E1 282.299} C_DIS
LIN {X 0.040,Y -444.160,Z 515.561,A 0.000,B 0.000,C 90.000,E1 280.950} C_DIS
LIN {X 0.002,Y -452.944,Z 515.555,A 0.000,B 0.000,C 90.000,E1 279.905} C_DIS
LIN {X -0.203,Y -459.023,Z 515.551,A 0.000,B 0.000,C 90.000,E1 279.151} C_DIS
LIN {X 0.106,Y -464.544,Z 515.546,A 0.000,B 0.000,C 90.000,E1 278.341} C_DIS
LIN {X -0.155,Y -471.123,Z 515.541,A 0.000,B 0.000,C 90.000,E1 277.352} C_DIS
LIN {X 0.061,Y -476.741,Z 515.535,A 0.000,B 0.000,C 90.000,E1 276.315} C_DIS
LIN {X 0.007,Y -480.383,Z 515.531,A 0.000,B 0.000,C 90.000,E1 275.568} C_DIS
LIN {X 0.166,Y -482.454,Z 515.528,A 0.000,B 0.000,C 90.000,E1 275.049} C_DIS
LIN {X -0.145,Y -484.207,Z 515.525,A 0.000,B 0.000,C 90.000,E1 274.588} C_DIS
LIN {X -0.006,Y -485.600,Z 515.523,A 0.000,B 0.000,C 90.000,E1 274.073} C_DIS
LIN {X 0.180,Y -486.675,Z 515.520,A 0.000,B 0.000,C 90.000,E1 273.555} C_DIS
LIN {X -0.116,Y -487.413,Z 515.517,A 0.000,B 0.000,C 90.000,E1 273.094} C_DIS
LIN {X 0.053,Y -487.823,Z 515.514,A 0.000,B 0.000,C 90.000,E1 272.579} C_DIS
LIN {X 0.231,Y -487.855,Z 515.512,A 0.000,B 0.000,C 90.000,E1 272.064} C_DIS
LIN {X -0.060,Y -487.534,Z 515.509,A 0.000,B 0.000,C 90.000,E1 271.604} C_DIS
LIN {X 0.120,Y -486.857,Z 515.506,A 0.000,B 0.000,C 90.000,E1 271.088} C_DIS
LIN {X -0.186,Y -485.657,Z 515.503,A 0.000,B 0.000,C 90.000,E1 270.630} C_DIS
LIN {X -0.010,Y -483.908,Z 515.501,A 0.000,B 0.000,C 90.000,E1 270.115} C_DIS
LIN {X 0.158,Y -481.507,Z 515.498,A 0.000,B 0.000,C 90.000,E1 269.599} C_DIS
LIN {X -0.006,Y -480.100,Z 515.497,A 0.000,B 0.000,C 90.000,E1 269.370} C_DIS
LIN {X -0.170,Y -478.438,Z 515.495,A 0.000,B 0.000,C 90.000,E1 269.141} C_DIS
LIN {X -0.035,Y -474.431,Z 515.492,A 0.000,B 0.000,C 90.000,E1 268.625} C_DIS
LIN {X -0.215,Y -472.071,Z 515.491,A 0.000,B 0.000,C 90.000,E1 268.396} C_DIS
LIN {X 0.054,Y -466.582,Z 515.488,A 0.000,B 0.000,C 90.000,E1 267.879} C_DIS
LIN {X 0.018,Y -463.505,Z 515.487,A 0.000,B 0.000,C 90.000,E1 267.650} C_DIS
LIN {X 0.197,Y -460.354,Z 515.486,A 0.000,B 0.000,C 90.000,E1 267.421} C_DIS
LIN {X -0.050,Y -453.433,Z 515.484,A 0.000,B 0.000,C 90.000,E1 267.078} C_DIS
LIN {X -0.175,Y -446.510,Z 515.482,A 0.000,B 0.000,C 90.000,E1 266.788} C_DIS
LIN {X 0.074,Y -439.564,Z 515.481,A 0.000,B 0.000,C 90.000,E1 266.502} C_DIS
LIN {X 0.203,Y -432.268,Z 515.479,A 0.000,B 0.000,C 90.000,E1 266.274} C_DIS
LIN {X -0.196,Y -424.078,Z 515.479,A 0.000,B 0.000,C 90.000,E1 266.159} C_DIS
LIN {X -0.211,Y -412.830,Z 515.478,A 0.000,B 0.000,C 90.000,E1 266.045} C_DIS
LIN {X 0.039,Y -407.479,Z 515.478,A 0.000,B 0.000,C 90.000,E1 265.988} C_DIS
LIN {X -0.018,Y -180.920,Z 515.478,A 0.000,B 0.000,C 90.000,E1 265.988} C_DIS
LIN {X 0.022,Y -180.852,Z 515.472,A 0.000,B 0.000,C 90.000,E1 264.951} C_DIS
LIN {X -0.078,Y -178.900,Z 515.443,A 0.000,B 0.000,C 90.000,E1 259.746} C_DIS
LIN {X 0.002,Y -175.944,Z 515.415,A 0.000,B 0.000,C 90.000,E1 254.629} C_DIS
LIN {X -0.051,Y -175.401,Z 515.410,A 0.000,B 0.000,C 90.000,E1 253.795} C_DIS
LIN {X -0.047,Y -172.169,Z 515.386,A 0.000,B 0.000,C 90.000,E1 249.518} C_DIS
LIN {X -0.008,Y -171.638,Z 515.381,A 0.000,B 0.000,C 90.000,E1 248.646} C_DIS
LIN {X -0.013,Y -167.861,Z 515.357,A 0.000,B 0.000,C 90.000,E1 244.332} C_DIS
LIN {X -0.070,Y -166.594,Z 515.348,A 0.000,B 0.000,C 90.000,E1 242.615} C_DIS
LIN {X 0.063,Y -162.584,Z 515.323,A 0.000,B 0.000,C 90.000,E1 238.201} C_DIS
LIN {X -0.100,Y -161.266,Z 515.314,A 0.000,B 0.000,C 90.000,E1 236.501} C_DIS
LIN {X 0.032,Y -157.267,Z 515.289,A 0.000,B 0.000,C 90.000,E1 232.029} C_DIS
LIN {X -0.042,Y -155.988,Z 515.279,A 0.000,B 0.000,C 90.000,E1 230.275} C_DIS
LIN {X -0.081,Y -152.244,Z 515.254,A 0.000,B 0.000,C 90.000,E1 225.810} C_DIS
LIN {X -0.058,Y -150.485,Z 515.239,A 0.000,B 0.000,C 90.000,E1 223.095} C_DIS
LIN {X -0.027,Y -147.209,Z 515.214,A 0.000,B 0.000,C 90.000,E1 218.543} C_DIS
LIN {X -0.057,Y -145.230,Z 515.194,A 0.000,B 0.000,C 90.000,E1 214.898} C_DIS
LIN {X 0.054,Y -142.354,Z 515.163,A 0.000,B 0.000,C 90.000,E1 209.333} C_DIS
LIN {X -0.019,Y -141.742,Z 515.153,A 0.000,B 0.000,C 90.000,E1 207.513} C_DIS
LIN {X 0.088,Y -139.489,Z 515.117,A 0.000,B 0.000,C 90.000,E1 200.972} C_DIS
LIN {X -0.055,Y -138.990,Z 515.101,A 0.000,B 0.000,C 90.000,E1 198.236} C_DIS
LIN {X 0.038,Y -138.335,Z 515.055,A 0.000,B 0.000,C 90.000,E1 189.792} C_DIS
LIN {X 0.062,Y -139.419,Z 515.008,A 0.000,B 0.000,C 90.000,E1 181.375} C_DIS
LIN {X -0.024,Y -141.337,Z 514.972,A 0.000,B 0.000,C 90.000,E1 174.894} C_DIS
LIN {X -0.067,Y -142.693,Z 514.956,A 0.000,B 0.000,C 90.000,E1 172.129} C_DIS
LIN {X 0.054,Y -145.057,Z 514.930,A 0.000,B 0.000,C 90.000,E1 167.465} C_DIS
LIN {X 0.050,Y -147.683,Z 514.910,A 0.000,B 0.000,C 90.000,E1 163.795} C_DIS
LIN {X -0.057,Y -150.329,Z 514.890,A 0.000,B 0.000,C 90.000,E1 160.188} C_DIS
LIN {X 0.014,Y -153.747,Z 514.870,A 0.000,B 0.000,C 90.000,E1 156.538} C_DIS
LIN {X 0.005,Y -157.160,Z 514.850,A 0.000,B 0.000,C 90.000,E1 152.948} C_DIS
LIN {X -0.061,Y -161.312,Z 514.830,A 0.000,B 0.000,C 90.000,E1 149.410} C_DIS
LIN {X -0.044,Y -164.427,Z 514.815,A 0.000,B 0.000,C 90.000,E1 146.755} C_DIS
LIN {X -0.048,Y -169.112,Z 514.796,A 0.000,B 0.000,C 90.000,E1 143.256} C_DIS
LIN {X -0.098,Y -171.665,Z 514.786,A 0.000,B 0.000,C 90.000,E1 141.537} C_DIS
LIN {X -0.052,Y -176.632,Z 514.767,A 0.000,B 0.000,C 90.000,E1 138.081} C_DIS
LIN {X 0.075,Y -180.930,Z 514.753,A 0.000,B 0.000,C 90.000,E1 135.486} C_DIS
LIN {X -0.061,Y -186.348,Z 514.734,A 0.000,B 0.000,C 90.000,E1 132.162} C_DIS
LIN {X 0.005,Y -190.981,Z 514.720,A 0.000,B 0.000,C 90.000,E1 129.644} C_DIS
LIN {X 0.103,Y -192.404,Z 514.715,A 0.000,B 0.000,C 90.000,E1 128.749} C_DIS
LIN {X 0.101,Y -290.120,Z 514.715,A 0.000,B 0.000,C 90.000,E1 128.749} C_DIS
LIN {X -0.007,Y -291.206,Z 514.715,A 0.000,B 0.000,C 90.000,E1 128.749} C_DIS
LIN {X 0.083,Y -295.310,Z 514.714,A 0.000,B 0.000,C 90.000,E1 128.543} C_DIS
LIN {X -0.057,Y -297.633,Z 514.713,A 0.000,B 0.000,C 90.000,E1 128.382} C_DIS
LIN {X -0.108,Y -300.816,Z 514.711,A 0.000,B 0.000,C 90.000,E1 128.016} C_DIS
LIN {X 0.128,Y -302.773,Z 514.709,A 0.000,B 0.000,C 90.000,E1 127.649} C_DIS
LIN {X -0.061,Y -304.301,Z 514.708,A 0.000,B 0.000,C 90.000,E1 127.363} C_DIS
LIN {X -0.046,Y -305.537,Z 514.706,A 0.000,B 0.000,C 90.000,E1 127.030} C_DIS
LIN {X 0.087,Y -316.465,Z 514.686,A 0.000,B 0.000,C 90.000,E1 123.420} C_DIS
LIN {X 0.098,Y -326.730,Z 514.670,A 0.000,B 0.000,C 90.000,E1 120.541} C_DIS
LIN {X 0.082,Y -338.343,Z 514.654,A 0.000,B 0.000,C 90.000,E1 117.719} C_DIS
LIN {X 0.080,Y -351.406,Z 514.639,A 0.000,B 0.000,C 90.000,E1 114.951} C_DIS
LIN {X -0.078,Y -364.335,Z 514.625,A 0.000,B 0.000,C 90.000,E1 112.567} C_DIS
LIN {X 0.148,Y -378.596,Z 514.612,A 0.000,B 0.000,C 90.000,E1 110.174} C_DIS
LIN {X 0.130,Y -394.296,Z 514.599,A 0.000,B 0.000,C 90.000,E1 107.873} C_DIS
LIN {X -0.123,Y -411.549,Z 514.587,A 0.000,B 0.000,C 90.000,E1 105.662} C_DIS
LIN {X -0.071,Y -430.478,Z 514.575,A 0.000,B 0.000,C 90.000,E1 103.467} C_DIS
LIN {X -0.212,Y -450.564,Z 514.563,A 0.000,B 0.000,C 90.000,E1 101.422} C_DIS
LIN {X 0.043,Y -471.203,Z 514.553,A 0.000,B 0.000,C 90.000,E1 99.500} C_DIS
LIN {X -0.197,Y -478.968,Z 514.549,A 0.000,B 0.000,C 90.000,E1 98.859} C_DIS
LIN {X -0.123,Y -480.956,Z 514.548,A 0.000,B 0.000,C 90.000,E1 98.624} C_DIS
LIN {X -0.121,Y -482.479,Z 514.547,A 0.000,B 0.000,C 90.000,E1 98.398} C_DIS
LIN {X 0.237,Y -483.758,Z 514.545,A 0.000,B 0.000,C 90.000,E1 98.106} C_DIS
LIN {X 0.113,Y -484.700,Z 514.544,A 0.000,B 0.000,C 90.000,E1 97.871} C_DIS
LIN {X -0.183,Y -485.736,Z 514.541,A 0.000,B 0.000,C 90.000,E1 97.409} C_DIS
LIN {X 0.006,Y -485.775,Z 514.538,A 0.000,B 0.000,C 90.000,E1 96.891} C_DIS
LIN {X 0.201,Y -484.823,Z 514.536,A 0.000,B 0.000,C 90.000,E1 96.372} C_DIS
LIN {X -0.084,Y -482.711,Z 514.533,A 0.000,B 0.000,C 90.000,E1 95.910} C_DIS
LIN {X 0.227,Y -481.079,Z 514.531,A 0.000,B 0.000,C 90.000,E1 95.625} C_DIS
LIN {X 0.140,Y -459.367,Z 514.516,A 0.000,B 0.000,C 90.000,E1 92.865} C_DIS
LIN {X 0.153,Y -448.898,Z 514.507,A 0.000,B 0.000,C 90.000,E1 91.318} C_DIS
LIN {X -0.106,Y -436.050,Z 514.496,A 0.000,B 0.000,C 90.000,E1 89.255} C_DIS
LIN {X 0.083,Y -424.664,Z 514.485,A 0.000,B 0.000,C 90.000,E1 87.364} C_DIS
LIN {X 0.177,Y -411.867,Z 514.473,A 0.000,B 0.000,C 90.000,E1 85.179} C_DIS
LIN {X 0.052,Y -397.789,Z 514.460,A 0.000,B 0.000,C 90.000,E1 82.704} C_DIS
LIN {X 0.002,Y -386.833,Z 514.449,A 0.000,B 0.000,C 90.000,E1 80.735} C_DIS
LIN {X -0.204,Y -375.827,Z 514.437,A 0.000,B 0.000,C 90.000,E1 78.757} C_DIS
LIN {X -0.122,Y -365.036,Z 514.426,A 0.000,B 0.000,C 90.000,E1 76.700} C_DIS
LIN {X 0.115,Y -353.851,Z 514.413,A 0.000,B 0.000,C 90.000,E1 74.283} C_DIS
LIN {X 0.019,Y -345.182,Z 514.401,A 0.000,B 0.000,C 90.000,E1 72.181} C_DIS
LIN {X 0.141,Y -332.102,Z 514.380,A 0.000,B 0.000,C 90.000,E1 68.465} C_DIS
LIN {X -0.035,Y -322.123,Z 514.363,A 0.000,B 0.000,C 90.000,E1 65.357} C_DIS
LIN {X 0.038,Y -314.320,Z 514.349,A 0.000,B 0.000,C 90.000,E1 62.794} C_DIS
LIN {X 0.111,Y -308.530,Z 514.338,A 0.000,B 0.000,C 90.000,E1 60.845} C_DIS
LIN {X 0.024,Y -300.807,Z 514.324,A 0.000,B 0.000,C 90.000,E1 58.250} C_DIS
LIN {X -0.183,Y -291.516,Z 514.305,A 0.000,B 0.000,C 90.000,E1 54.975} C_DIS
LIN {X -0.119,Y -284.506,Z 514.290,A 0.000,B 0.000,C 90.000,E1 52.271} C_DIS
LIN {X 0.049,Y -279.060,Z 514.279,A 0.000,B 0.000,C 90.000,E1 50.194} C_DIS
LIN {X -0.098,Y -275.185,Z 514.271,A 0.000,B 0.000,C 90.000,E1 48.852} C_DIS
LIN {X -0.112,Y -271.023,Z 514.264,A 0.000,B 0.000,C 90.000,E1 47.472} C_DIS
LIN {X 0.128,Y -264.259,Z 514.252,A 0.000,B 0.000,C 90.000,E1 45.324} C_DIS
LIN {X -0.082,Y -254.900,Z 514.236,A 0.000,B 0.000,C 90.000,E1 42.528} C_DIS
